METHOD M_PT100_Interpolate_Ohm2C : LREAL
VAR_INPUT
	in_lrOhm:	LREAL;	// Resistance reading [Ohm]
	// Index of the first lookup table entry with 
	// value lower than the measured resistance.
	in_nIndex:	INT;	
END_VAR
VAR
	lrR1, lrR2:	LREAL;	// Temporary variables
END_VAR
IF in_nIndex = 0 OR in_nIndex = 88	THEN
	M_PT100_Interpolate_Ohm2C	:= LookupTable[in_nIndex].celsius;
ELSE
	// Linear interpolation Example
	//	Index 8		(celsius := 	-200.0	, ohm := 	18.522	),
	//  Reading                               ohm := 	20.123
	//	Index 9		(celsius := 	-195.0	, ohm := 	20.679	),
	//
	//   TempC = -200.0 + (20.123-18.522) / (20.679-18.522) * 5.0 
	//         = -200.0 + 1.601 / 2.157 * 5.0
	//         = -196.289 degC

	lrR1	:= in_lrOhm - LookupTable[in_nIndex].ohm;
	lrR2	:= LookupTable[in_nIndex+1].ohm - LookupTable[in_nIndex].ohm;
	M_PT100_Interpolate_Ohm2C	:= LookupTable[in_nIndex].celsius + lrR1/lrR2 * lrTemStep;
END_IF
END_METHOD

// Convert raw resistance reading [bit] (Ohm*64) to degrees Celsius.
// The input value has to be devided by 64 to get the reading in [Ohm].
METHOD M_PT100_Ohm2C : LREAL
VAR_INPUT
	in_lrOhmRaw:	INT;	// Raw reading [bit]. [Ohm] = in_lrOhmRaw/64
END_VAR
VAR
	i:		INT;
	lrOhm:	LREAL; 	// PT100 Resistance reading [Ohm]
END_VAR
// Raw reading of -1 means a broken wire or failed sensor.
// The convention is to return 850 degC
IF in_lrOhmRaw	= -1	THEN
	M_PT100_Ohm2C	:= 850.0;
	RETURN;
END_IF

// Get reading in [Ohm]
lrOhm	:= INT_TO_LREAL(in_lrOhmRaw) / 64.0;


// Find the first index in the table
// where the resistance value is lower that the reading.

IF lrOhm > LookupTable[nLastIndex].ohm	THEN
	// We are increasing the index until we find a reading in the
	// table that is higher than the measurement
	FOR i := nLastIndex TO 88	DO
		IF i = 88	THEN
			// We are at the highest temperature in the lookup table.
			// Take that value;
			M_PT100_Ohm2C	:= LookupTable[i].celsius;
			RETURN;
		ELSE
			IF lrOhm < LookupTable[i].ohm	THEN
				// We crossed the correct reading.
				// Remember the index for faster next reading.
				nLastIndex	:= i-1;
				IF nLastIndex < 0	THEN
					nLastIndex	:= 0;
				END_IF
				M_PT100_Ohm2C	:= M_PT100_Interpolate_Ohm2C(lrOhm,nLastIndex);
				RETURN;
			ELSIF lrOhm = LookupTable[i].ohm	THEN
				// We crossed the correct reading.
				// Remember the index for faster next reading.
				nLastIndex	:= i;
				M_PT100_Ohm2C	:= M_PT100_Interpolate_Ohm2C(lrOhm,nLastIndex);
				RETURN;
			END_IF
		END_IF
	END_FOR
ELSIF lrOhm < LookupTable[nLastIndex].ohm	THEN
	// We are decreasing the index until we find a reading in the
	// table that is higher than the measurement
	FOR i := nLastIndex TO 0 BY  -1	DO
		IF i <= 0	THEN
			// We are at the lowest temperature in the lookup table.
			// Take that value;
			M_PT100_Ohm2C	:= LookupTable[0].celsius;
			RETURN;
		ELSE
			IF lrOhm > LookupTable[i].ohm	THEN
				// We crossed the correct reading.
				// Remember the index for faster next reading.
				nLastIndex	:= i;
				M_PT100_Ohm2C	:= M_PT100_Interpolate_Ohm2C(lrOhm,nLastIndex);
				RETURN;
			ELSIF lrOhm = LookupTable[i].ohm	THEN
				// We crossed the correct reading.
				// Remember the index for faster next reading.
				nLastIndex	:= i;
				M_PT100_Ohm2C	:= M_PT100_Interpolate_Ohm2C(lrOhm,nLastIndex);
				RETURN;
			END_IF
		END_IF
	END_FOR
ELSE
	M_PT100_Ohm2C	:= M_PT100_Interpolate_Ohm2C(lrOhm,nLastIndex);
	RETURN;
END_IF
END_METHOD

// Calculate pressure based on the status in input value
METHOD M_SetStatus
VAR_INPUT
END_VAR
VAR
END_VAR
// Set temperature sensor type
stat.nType	:= in_nType;

// Update value depending on the sensor type.
// So far, only PT100 supported.
CASE in_nType OF
	E_CRYO_SENSOR_TYPE_TEMP.PT100:
		M_SetStatus_PT100();
END_CASE
END_METHOD

// Calculate pressure based on the status in input value
METHOD M_SetStatus_PT100
VAR_INPUT
END_VAR
VAR
END_VAR
//
// Set the temperature as it is read.
// Later on we decide if it is valid or not.
//
IF NOT in_bResistor_1_64	THEN
	// Standard RTD reading
	stat.lrTempC	:= i_nValue * in_lrScale;	// Set temperature in deg C
	stat.lrTempK	:= stat.lrTempC + 273.15;	// Set temperature in deg K
ELSE	
	// RTD reading of resistance.
	// i_nValue is in [Ohm]
	stat.lrTempC	:= M_PT100_Ohm2C(i_nValue);	// Set temperature in deg C
	stat.lrTempK	:= stat.lrTempC + 273.15;	// Set temperature in deg K
END_IF

// Reading in Celsius of 850.0 means an error.
// In this case, set the Kelvin reading to 850.0 as well.
// Set error and not Valid and return.
IF stat.lrTempC = 850.0	THEN
	stat.lrTempK	:= 850.0;
	stat.bError		:= TRUE;
	stat.bValid		:= FALSE;
	RETURN;
END_IF

//
// Update validity
// Note: bInputError = (bInputUnder OR bInputOver)
//       bValid      = TRUE if PDO is OK (nothing to do with bError)
//
IF stat.bInputActive THEN
	IF stat.bInputError  AND  stat.bInputUnder  AND  in_bIgnoreUnderrange 	THEN
		// Sometimes we ignore underrange because PT100 cannot read below -200C.
		// The bUnderrange flag is still active!!!
		stat.bError	:= FALSE;
		stat.bValid	:= TRUE;
	ELSIF stat.bInputError 	THEN
		stat.bError	:= TRUE;
		stat.bValid	:= FALSE;
	ELSE
		stat.bError	:= FALSE;
		stat.bValid	:= TRUE;
	END_IF
ELSE
	stat.bError	:= TRUE;
	stat.bValid	:= FALSE;
END_IF
END_METHOD

END_FUNCTION_BLOCK

// ---- POUs/Simulation/FB_CRYO_SIM_CTRL.TcPOU
FUNCTION_BLOCK FB_CRYO_SIM_CTRL
VAR_INPUT
	in_ptr_Cryo_Ctrl:	POINTER TO FB_CRYO_CTRL;
END_VAR
VAR
	{attribute 'OPC.UA.DA' := '1'}
	SIM_Temp_Mirror:		FB_CRYO_SIM_TEMPERATURE;

	{attribute 'OPC.UA.DA' := '1'}
	SIM_Temp_LN2_Exhaust:	FB_CRYO_SIM_TEMPERATURE;
	
	{attribute 'OPC.UA.DA' := '1'}
	SIM_Temp_LN2_Inlet:		FB_CRYO_SIM_TEMPERATURE;
	
	{attribute 'OPC.UA.DA' := '1'}
	SIM_Temp_DET:			FB_CRYO_SIM_TEMPERATURE;
	
	{attribute 'OPC.UA.DA' := '1'}
	SIM_Pressure_Cryo:	FB_CRYO_SIM_PRESSURE;		// Cryo Pressure simulator
	
	{attribute 'OPC.UA.DA' := '1'}
	SIM_Pressure_Evac:	FB_CRYO_SIM_PRESSURE;		// Evacuation Pressure simulator
	
	
	
	{attribute 'OPC.UA.DA' := '1'}
	nCryoState:		E_CRYO_CTRL_STATE	:= E_CRYO_CTRL_STATE.NONE;
	{attribute 'OPC.UA.DA' := '0'}
	nCryoOldState:	E_CRYO_CTRL_STATE	:= E_CRYO_CTRL_STATE.NONE;
	
	{attribute 'OPC.UA.DA' := '0'}
	trgCMD:			R_TRIG;
	{attribute 'OPC.UA.DA' := '0'}
	trgEvacOn:		R_TRIG;
	{attribute 'OPC.UA.DA' := '0'}
	trgEvacOff:		F_TRIG;
	{attribute 'OPC.UA.DA' := '0'}
	trgInVacuum:	R_TRIG;
	{attribute 'OPC.UA.DA' := '0'}
	trgPrecoolOff:	F_TRIG;
	{attribute 'OPC.UA.DA' := '0'}
	trgCoolOff:		F_TRIG;
	{attribute 'OPC.UA.DA' := '0'}
	trgWarmupOff:	F_TRIG;
	
	nRampPeriod:	UDINT := 20000;
	
	{attribute 'OPC.UA.DA' := '0'}
	lrTmp:	LREAL;
	
	
END_VAR

//
// Get Cryo controller State
//
nCryoState	:= in_ptr_Cryo_Ctrl^.stat.nState;


//
// Execute simulators for all temperatures and pressures, etc.
//
SIM_Temp_Mirror(
	in_lrScale		:= in_ptr_Cryo_Ctrl^.Temp_Mirror.in_lrScale_1, 
	in_lrTempK		:= );
	
SIM_Temp_LN2_Exhaust(
	in_lrScale		:= in_ptr_Cryo_Ctrl^.Temp_LN2_Exhaust.in_lrScale_1, 
	in_lrTempK		:= 88.75,	//	Variation 88.75 +- 11.25, i.e. [77.50..100.00]
	in_lrTempDelta	:= 11.25,
	in_nPeriod		:= 10000,
	in_bAutoSine	:= TRUE);
	
SIM_Temp_LN2_Inlet(
	in_lrScale		:= in_ptr_Cryo_Ctrl^.Temp_LN2_Inlet.in_lrScale_1, 
	in_lrTempK		:= 77.15);
	
SIM_Temp_DET(
	in_lrScale		:= in_ptr_Cryo_Ctrl^.Temp_DET.in_lrScale_1, 
	in_lrTempK		:= );
	
SIM_Pressure_Cryo(
	in_nType		:= in_ptr_Cryo_Ctrl^.Pressure_Cryo.in_nType_1,
	in_lrBitsPerVolt:= in_ptr_Cryo_Ctrl^.Pressure_Cryo.in_lrBitsPerVolt_1, 
	in_nPeriod		:= nRampPeriod);
	
SIM_Pressure_Evac(
	in_nType		:= in_ptr_Cryo_Ctrl^.Pressure_Evac.in_nType_1,
	in_lrBitsPerVolt:= in_ptr_Cryo_Ctrl^.Pressure_Evac.in_lrBitsPerVolt_1, 
	in_nPeriod		:= nRampPeriod);


	
	
//	
// Capture Cryo controller change of state.
//
trgCMD(CLK:=(nCryoState<>nCryoOldState));
nCryoOldState	:= nCryoState;

// NOTE: This code is execute only once on each State change.
IF trgCMD.Q  THEN
	// The state of Cryo controller has changed.
	// Take action with simulators.
	CASE nCryoState OF
		
		/////////////////////////////////
		E_CRYO_CTRL_STATE.PRE_COOLING:
		/////////////////////////////////
		//
		// Trigger Bench temperature ramp 1 K below PRE_COOL threshold
		SIM_Temp_Mirror.M_RampTo(
			in_lrValueEnd	:= in_ptr_Cryo_Ctrl^.cfg.lrTemp_Precooled-1.0,
			in_nPeriod		:= nRampPeriod);

		// Trigger DET temperature ramp 1 K below PRE_COOL threshold.
		// Slow down the ramp compared to the Bench, so
		// DET temperature is slightly higher during cooldown.
		// The final temperature is the same as for the Bench.
		SIM_Temp_DET.M_RampTo(
			in_lrValueEnd	:= in_ptr_Cryo_Ctrl^.cfg.lrTemp_Precooled-1.0,
			in_nPeriod		:= nRampPeriod + 5000);
			
		/////////////////////////////////
		E_CRYO_CTRL_STATE.COOLING_DOWN:
		/////////////////////////////////
		//
		// Trigger temperature ramp 1 K below COOL threshold
		SIM_Temp_Mirror.M_RampTo(
			in_lrValueEnd	:= in_ptr_Cryo_Ctrl^.cfg.lrTemp_Cold-1.0,
			in_nPeriod		:= nRampPeriod);
			
		// Trigger temperature ramp 1 K below COOL threshold
		// Slow down the ramp compared to the Bench, so
		// DET temperature is slightly higher during cooldown.
		// The final temperature is the same as for the Bench.
		SIM_Temp_DET.M_RampTo(
			in_lrValueEnd	:= in_ptr_Cryo_Ctrl^.cfg.lrTemp_Cold-1.0,
			in_nPeriod		:= nRampPeriod + 5000);
			
		/////////////////////////////////
		E_CRYO_CTRL_STATE.WARMING_UP:
		/////////////////////////////////
		//
		// Trigger temperature ramp to in_ptr_Cryo_Ctrl^.cfg.lrTemp_Warm (~10C)
		SIM_Temp_Mirror.M_RampTo(
			in_lrValueEnd	:= in_ptr_Cryo_Ctrl^.cfg.lrTemp_Warm + 1.0,
			in_nPeriod		:= nRampPeriod);
			
			
		// Trigger temperature ramp to in_ptr_Cryo_Ctrl^.cfg.lrTemp_Warm (~10C)
		// Speed up the ramp compared to the Bench, so
		// DET temperature is slightly higher during warm-up.
		// The final temperature is the same as for the Bench.
		SIM_Temp_DET.M_RampTo(
			in_lrValueEnd	:= in_ptr_Cryo_Ctrl^.cfg.lrTemp_Warm + 1.0,
			in_nPeriod		:= nRampPeriod - 2000);
			
		/////////////////////////////////
		E_CRYO_CTRL_STATE.REPRESSURIZING:
		/////////////////////////////////
		//
		// Trigger Cryo vacuum ramp to atmospheric pressure ~820 mbar
		SIM_Pressure_Cryo.M_RampTo(
			in_lrValueEnd	:= 820.0,
			in_nPeriod		:= 17000);
			
		// Follow the same ramp with Evac but a bit slower.
		SIM_Pressure_Evac.M_RampTo(
			in_lrValueEnd	:= 820.0,
			in_nPeriod		:= 20000);
	END_CASE

END_IF


//
// Evacuation Pressure simulation
//
// Capture Evacuation ON/OFF trigger
trgEvacOn(CLK := in_ptr_Cryo_Ctrl^.ctrl.bEnable_Evac);
trgEvacOff(CLK := in_ptr_Cryo_Ctrl^.ctrl.bEnable_Evac);
IF	trgEvacOn.Q THEN
	// Trigger vacuum ramp 0.0001 mbar below Good Vacuum
	SIM_Pressure_Cryo.M_StartCurve(
		in_lrValueEnd	:= in_ptr_Cryo_Ctrl^.Pressure_Cryo.in_lrLimitGoodVac - 0.0001, 
		in_nPeriod		:= 20000, 
		in_lrCurveScale	:= 0.3);
ELSIF trgEvacOff.Q THEN
	// Evacuation stopped.
	// Keep the pressure as it is.
	SIM_Pressure_Cryo.M_Stop();
END_IF


//
// If Turbo Pump is running, keep Evacuation pressure 1.0e-05 below the Cryo pressure.
// Value is calculated on every cycle.
//
IF in_ptr_Cryo_Ctrl^.EvacSys.stat.bTurboPumpON THEN
	SIM_Pressure_Evac.M_SetValue(SIM_Pressure_Cryo.lrPress - 1.0E-05);
END_IF


//
// To get more realistic evacuation,
// Restart simulated curve when inVacuum is triggered.
//
//trgInVacuum(CLK := in_ptr_Cryo_Ctrl^.Pressure_Cryo.stat.bInVacuum);
trgInVacuum(CLK := in_ptr_Cryo_Ctrl^.stat.bInVacuum);
IF trgInVacuum.Q THEN
	SIM_Pressure_Cryo.M_StartCurve(
		in_lrValueEnd	:= in_ptr_Cryo_Ctrl^.Pressure_Cryo.in_lrLimitGoodVac - 0.0001, 
		in_nPeriod		:= 10000, 
		in_lrCurveScale	:= 0.3);
END_IF

			
//
// Capture events when buttons are released 
// and temperature transitions interrupted.
//

// Capture pre-cooling, cooling or warmup button release.
// Stop ramping in that case.
trgPrecoolOff	(CLK:=in_ptr_Cryo_Ctrl^.ctrl.bEnable_Precool);
trgCoolOff		(CLK:=in_ptr_Cryo_Ctrl^.ctrl.bEnable_Cool);
trgWarmupOff	(CLK:=in_ptr_Cryo_Ctrl^.ctrl.bEnable_Warmup);

IF	trgPrecoolOff.Q OR trgCoolOff.Q OR trgWarmupOff.Q	THEN
	SIM_Temp_Mirror.M_Stop();
	SIM_Temp_DET.M_Stop();
END_IF

END_FUNCTION_BLOCK

// ---- POUs/Simulation/FB_CRYO_SIM_TEMPERATURE.TcPOU
//
// This FB simulates temperature in degK.
//
FUNCTION_BLOCK FB_CRYO_SIM_TEMPERATURE
VAR_INPUT
	in_lrScale:		LREAL 	:= 0.1;		// Scale factor, T = raw * scale. Default 0.1
	in_lrTempK:		LREAL	:= 283.15;	// Start Temperature [K]
	in_lrTempDelta:	LREAL	:= 11.25;	// Delta Temperature +- for SINE wave [K]
	in_nPeriod:		UDINT	:= 10000;	// RAMP/SINE Command period, default 10000ms = 10s
	in_bAutoSine:	BOOL	:= FALSE;	// Flag if SINE wave should start immediately
	
END_VAR
VAR
	q_nStatus	AT%Q*:	UINT	:= 0;	// Simulated status
	q_nValue	AT%Q*:	INT		:= 100;	// Simulated value [bit]
	
	{attribute 'OPC.UA.DA' := '0'}
	bStarted:		BOOL := FALSE;
	{attribute 'OPC.UA.DA' := '0'}
	toggleTimer:	TON;		// Timer for PDO (alive) toggle
	{attribute 'OPC.UA.DA' := '0'}
	rampTimer:		TON;		// Timer for temperature ramp

	{attribute 'OPC.UA.DA' := '0'}
	nToggleMask:	UINT := 2#1000_0000_0000_0000;

	lrTempK:		LREAL	:= 283.15;	// Simulated temperature [K]
	{attribute 'OPC.UA.DA' := '0'}
	lrTempStart:	LREAL	:= 283.15;	// Simulated temperature start [K]
	{attribute 'OPC.UA.DA' := '0'}
	lrTempEnd:		LREAL	:= 0.0;		// Simulated temperature end   [K]
	{attribute 'OPC.UA.DA' := '0'}
	lrTempDelta:	LREAL	:= 11.25;	// Delta Temperature +- for SINE wave [K]
	{attribute 'OPC.UA.DA' := '0'}
	nValue:			INT		:= 100;		// Simulated value [bit]

	{attribute 'OPC.UA.DA' := '0'}
	nPeriod:		UDINT	:= 10000;	// RAMP/SINE Command period, default 10000ms = 10s
	
	{attribute 'OPC.UA.DA' := '0'}
	nState:		INT	:= SIM_TEMP_STATE_FIXED;
	
END_VAR
VAR CONSTANT 
	{attribute 'OPC.UA.DA' := '0'}
    SIM_TEMP_STATE_NONE:	INT :=  0;
	{attribute 'OPC.UA.DA' := '0'}
    SIM_TEMP_STATE_FIXED:	INT := 10;
	{attribute 'OPC.UA.DA' := '0'}
    SIM_TEMP_STATE_RAMP:	INT := 20;
	{attribute 'OPC.UA.DA' := '0'}
    SIM_TEMP_STATE_SINE:	INT := 30;
	
	{attribute 'OPC.UA.DA' := '0'}
    SIM_TEMP_RAMP_UP:		INT := 0;
	{attribute 'OPC.UA.DA' := '0'}
    SIM_TEMP_RAMP_DOWN:		INT := 1;
	
END_VAR

//
// Simulate terminal alive toggle every 160ms.
//
IF NOT bStarted THEN
	bStarted	:= TRUE;
	lrTempK		:= in_lrTempK;	// Assign starting value
	lrTempDelta	:= in_lrTempDelta;
	nPeriod		:= in_nPeriod;
	IF in_bAutoSine THEN
		M_StartSine(in_lrValueStart:=lrTempK,
					in_lrValueDelta:=lrTempDelta,
					in_nPeriod:=nPeriod);
	END_IF
	toggleTimer(IN:=FALSE);
END_IF
toggleTimer(IN:=TRUE,PT:=T#160MS);

IF toggleTimer.Q THEN
	q_nStatus	:= q_nStatus XOR nToggleMask;
	// Restart the timer
	toggleTimer(IN:=FALSE);
END_IF


//
// Handle states 
//
IF nState = SIM_TEMP_STATE_RAMP THEN
	rampTimer(IN:=TRUE);
	lrTempK	:=	lrTempStart + 
				(lrTempEnd - lrTempStart)* TIME_TO_LREAL(rampTimer.ET)/TIME_TO_LREAL(rampTimer.PT);
	IF rampTimer.Q THEN
		rampTimer(IN:=FALSE);
		nState	:= SIM_TEMP_STATE_FIXED;
	END_IF
ELSIF nState = SIM_TEMP_STATE_SINE THEN
	rampTimer(IN:=TRUE);
	lrTempK	:=	lrTempStart + 
				lrTempDelta * SIN(2 * PI * TIME_TO_LREAL(rampTimer.ET)/TIME_TO_LREAL(rampTimer.PT));
	IF rampTimer.Q THEN
		rampTimer(IN:=FALSE);
		// Continue with the sine wave.
		rampTimer(IN:=TRUE,PT:=UDINT_TO_TIME(nPeriod));
	END_IF
END_IF



//
// Set the raw reading, i.e. K -> bit.
//
q_nValue	:= M_degK2bit(lrTempK);

METHOD M_bit2degK : LREAL
VAR_INPUT
	in_nValue:	INT;
END_VAR
//
// Set the raw reading, i.e. K -> bit.
// Conversion is K -> C -> bit.
//
M_bit2degK	:= in_nValue * in_lrScale + 273.15;
END_METHOD

METHOD M_degK2bit : INT
VAR_INPUT
	in_lrValue:	LREAL;
END_VAR
//
// Set the raw reading, i.e. K -> bit.
// Conversion is K -> C -> bit.
//
M_degK2bit	:= LREAL_TO_INT((in_lrValue - 273.15) / in_lrScale);
END_METHOD

METHOD M_RampTo
VAR_INPUT
	in_lrValueEnd:		LREAL;
	in_nPeriod:			UDINT	:= 10000;	// RAMP/SINE Command period, default 10000ms = 10s
END_VAR
rampTimer(IN:=FALSE);
rampTimer(IN:=TRUE,PT:=UDINT_TO_TIME(in_nPeriod));
lrTempStart	:= lrTempK;
lrTempEnd	:= in_lrValueEnd;
nPeriod		:= in_nPeriod;
nState		:= SIM_TEMP_STATE_RAMP;
END_METHOD

METHOD M_SetValue
VAR_INPUT
	in_lrValue:	LREAL;
END_VAR
rampTimer(IN:=FALSE);
lrTempK	:= in_lrValue;
nState	:= SIM_TEMP_STATE_FIXED;
END_METHOD

METHOD M_StartRamp
VAR_INPUT
	in_lrValueStart:	LREAL;
	in_lrValueEnd:		LREAL;
	in_nPeriod:			UDINT	:= 10000;	// RAMP/SINE Command period, default 10000ms = 10s
END_VAR
rampTimer(IN:=FALSE);
rampTimer(IN:=TRUE,PT:=UDINT_TO_TIME(in_nPeriod));
lrTempStart	:= in_lrValueStart;
lrTempEnd	:= in_lrValueEnd;
nPeriod		:= in_nPeriod;
nState		:= SIM_TEMP_STATE_RAMP;
END_METHOD

METHOD M_StartSine
VAR_INPUT
	in_lrValueStart:	LREAL;
	in_lrValueDelta:	LREAL;
	in_nPeriod:			UDINT	:= 10000;	// RAMP/SINE Command period, default 10000ms = 10s
END_VAR
rampTimer(IN:=FALSE);
rampTimer(IN:=TRUE,PT:=UDINT_TO_TIME(in_nPeriod));
lrTempStart	:= in_lrValueStart;
lrTempDelta	:= in_lrValueDelta;
nPeriod		:= in_nPeriod;
nState		:= SIM_TEMP_STATE_SINE;
END_METHOD

METHOD M_Stop
VAR_INPUT
END_VAR
// Stop ramping.
// Keep value as it is.
rampTimer(IN:=FALSE);
nState	:= SIM_TEMP_STATE_FIXED;
END_METHOD

END_FUNCTION_BLOCK

// ---- POUs/Simulation/FB_CRYO_SIM_PRESSURE.TcPOU
//
// This FB simulates pressure.
//
FUNCTION_BLOCK FB_CRYO_SIM_PRESSURE
VAR_INPUT
	in_nType:	E_CRYO_SENSOR_TYPE_PRESS;
	// Scale factor bits -> Volt, U = raw / scale. 
	// Default for 16-bit, +-10V or 0..10V AI: 2^16/10/2 = 3276.8 bit
	in_lrBitsPerVolt:	LREAL := 3276.8;	// Scale factor, U = raw / scale. Default 3276.8
	in_lrPress:		LREAL	:= 777.0;	// Starting Pressure
	in_nPeriod:		UDINT	:= 10000;	// RAMP Command period, default 10000ms = 10s
	
END_VAR
VAR
	q_nStatus	AT%Q*:	UINT	:= 0;		// Simulated status
	q_nValue	AT%Q*:	INT		:= 27953;	// Simulated value [bit] = 777 mbar
	
	{attribute 'OPC.UA.DA' := '0'}
	bStarted:		BOOL := FALSE;
	{attribute 'OPC.UA.DA' := '0'}
	toggleTimer:	TON;		// Timer for PDO (alive) toggle
	{attribute 'OPC.UA.DA' := '0'}
	rampTimer:		TON;		// Timer for temperature ramp

	{attribute 'OPC.UA.DA' := '0'}
	nToggleMask:	UINT := 2#1000_0000_0000_0000;

	lrPress:		LREAL	:= 777.0;	// Simulated Pressure
	{attribute 'OPC.UA.DA' := '0'}
	lrPressStart:	LREAL	:= 0.0;		// Simulated Pressure start[mbar]
	{attribute 'OPC.UA.DA' := '0'}
	lrPressEnd:		LREAL	:= 0.0;		// Simulated Pressure end  [mbar]
	{attribute 'OPC.UA.DA' := '0'}
	lrPressDelta:	LREAL	:= 0.0;		// Simulated Pressure delta for curve  [mbar]
	{attribute 'OPC.UA.DA' := '0'}
	lrCurveScale:	LREAL	:= 0.3;		// t^lrCurveScale factor
	{attribute 'OPC.UA.DA' := '0'}
	nValue:			INT		:= 27953;	// Simulated value [bit]
	{attribute 'OPC.UA.DA' := '0'}
	nPeriod:		UDINT	:= 10000;	// RAMP Command period, default 10000ms = 10s
	
	{attribute 'OPC.UA.DA' := '0'}
	State:		INT	:= SIM_VACUUM_STATE_FIXED;
	
	// Temporary variables
	{attribute 'OPC.UA.DA' := '0'}
	lrTmp1:		LREAL;
	
END_VAR
VAR CONSTANT 
	{attribute 'OPC.UA.DA' := '0'}
    SIM_VACUUM_STATE_NONE:	INT :=  0;
	{attribute 'OPC.UA.DA' := '0'}
    SIM_VACUUM_STATE_FIXED:	INT := 10;
	{attribute 'OPC.UA.DA' := '0'}
    SIM_VACUUM_STATE_RAMP:	INT := 20;
	{attribute 'OPC.UA.DA' := '0'}
    SIM_VACUUM_STATE_CURVE:	INT := 30;
	
	{attribute 'OPC.UA.DA' := '0'}
    SIM_VACUUM_RAMP_UP:		INT := 0;
	{attribute 'OPC.UA.DA' := '0'}
    SIM_VACUUM_RAMP_DOWN:	INT := 1;
	
END_VAR

//
// Simulate terminal alive toggle every 160ms.
//
IF NOT bStarted THEN
	bStarted	:= TRUE;
	lrPress		:= in_lrPress;
	nPeriod		:= in_nPeriod;
	toggleTimer(IN:=FALSE);
END_IF
toggleTimer(IN:=TRUE,PT:=T#160MS);

IF toggleTimer.Q THEN
	q_nStatus	:= q_nStatus XOR nToggleMask;
	// Restart the timer
	toggleTimer(IN:=FALSE);
END_IF



//
// Handle states
//
rampTimer(IN:=TRUE);
IF State = SIM_VACUUM_STATE_RAMP THEN
	lrPress	:=	lrPressStart + 
				(lrPressEnd - lrPressStart)* TIME_TO_LREAL(rampTimer.ET)/TIME_TO_LREAL(rampTimer.PT);
	IF rampTimer.Q THEN
		rampTimer(IN:=FALSE);
		State	:= SIM_VACUUM_STATE_FIXED;
	END_IF
ELSIF State = SIM_VACUUM_STATE_CURVE THEN
	lrTmp1	:= TIME_TO_LREAL(rampTimer.ET)/TIME_TO_LREAL(rampTimer.PT);
	lrTmp1	:= EXPT(lrTmp1,lrCurveScale);
	lrPress	:=	lrPressStart + (lrPressEnd - lrPressStart)* lrTmp1;
	IF rampTimer.Q THEN
		rampTimer(IN:=FALSE);
		State	:= SIM_VACUUM_STATE_FIXED;
	END_IF
END_IF


//
// Set the raw reading, i.e. mbar -> bit.
// Conversion is mbar -> Volt -> bit.
//
IF lrPress > 0.0  THEN
	q_nValue	:= M_mbar2bit(lrPress);
END_IF

METHOD M_bit2mbar : LREAL
VAR_INPUT
	in_nBits:	INT;
END_VAR
VAR
	lrVoltage:	LREAL;
	lrPressure:	LREAL;
END_VAR
lrVoltage	:= in_nBits / in_lrBitsPerVolt;

CASE in_nType OF 
	E_CRYO_SENSOR_TYPE_PRESS.PKR_250,
	E_CRYO_SENSOR_TYPE_PRESS.PKR_360:
		// Conversion Volt -> mbar.
		// Pfeiffer PKR250/251
		// P = 10^(C1 * U - C2).
		// C1 = 1.667, C2 = d = 11.33
		// P = 10^(1.667 * U - 11.33)
		// U = (log(P)+C2)/C1
		// U = (log(P)+11.33)/1.667
		lrPressure	:= EXPT(10.0, (1.667 * lrVoltage - 11.33));
	E_CRYO_SENSOR_TYPE_PRESS.CMR_361:
		// Conversion Volt -> mbar.
		// Pfeiffer CMR361
		// P = (U - 1) * C1 * C2 [mbar]
		// C1 = 0.125, C2=FullScale = 1000 
		// P = (U - 1) * 0.125 * 1000.0 = (U-1) * 125[mbar]
		// P = (U-1) * 125
		// U = P/125 + 1
		lrPressure	:= (lrVoltage - 1) * 125;
	E_CRYO_SENSOR_TYPE_PRESS.WRG_D_NW25:
		// Edwards WRG-D-NW25 Conversion Volt -> mbar.
		// Range 10^-9 .. 100
		// P = 10^(C1 * U - C2).
		// P = 10^(1.5 * U - 12.0)
		// Valid range for U is 2.0-10.0
		lrPressure	:= EXPT(10.0, (1.5 * lrVoltage - 12.0));
END_CASE

M_bit2mbar	:= lrPressure;
END_METHOD

METHOD M_mbar2bit : INT
VAR_INPUT
	in_lrValue:	LREAL;
END_VAR
VAR
	lrValue:	LREAL;
	lrVoltage:	LREAL;
END_VAR
// Pressure cannot be zero
lrValue := MAX(1.0E-9,in_lrValue);

CASE in_nType OF 
	E_CRYO_SENSOR_TYPE_PRESS.PKR_250,
	E_CRYO_SENSOR_TYPE_PRESS.PKR_360:
		// Conversion Volt -> mbar.
		// Pfeiffer PKR250/251
		// P = 10^(C1 * U - C2).
		// C1 = 1.667, C2 = d = 11.33
		// P = 10^(1.667 * U - 11.33)
		// U = (log(P)+C2)/C1
		// U = (log(P)+11.33)/1.667
		lrVoltage	:= (LOG(lrValue) + 11.33) / 1.667;
	E_CRYO_SENSOR_TYPE_PRESS.CMR_361:
		// Conversion Volt -> mbar.
		// Pfeiffer CMR361
		// P = (U - 1) * C1 * C2 [mbar]
		// C1 = 0.125, C2=FullScale = 1000 
		// P = (U - 1) * 0.125 * 1000.0 = (U-1) * 125[mbar]
		// P = (U-1) * 125
		// U = P/125 + 1
		lrVoltage	:= lrValue/125 + 1.0;
	E_CRYO_SENSOR_TYPE_PRESS.WRG_D_NW25:
		// Edwards WRG-D-NW25 Conversion Volt -> mbar.
		// Range 10^-9 .. 100
		// P = 10^(C1 * U - C2).
		// P = 10^(1.5 * U - 12.0)
		// Valid range for U is 2.0-10.0
		lrVoltage	:= (LOG(lrValue) + 12.0) / 1.5;
END_CASE

M_mbar2bit	:= LREAL_TO_INT(lrVoltage * in_lrBitsPerVolt);
END_METHOD

METHOD M_RampTo
VAR_INPUT
	in_lrValueEnd:		LREAL;
	in_nPeriod:			UDINT	:= 10000;	// RAMP/SINE Command period, default 10000ms = 10s
END_VAR
rampTimer(IN:=FALSE);
rampTimer(IN:=TRUE,PT:=UDINT_TO_TIME(in_nPeriod));
lrPressStart	:= lrPress;
lrPressEnd		:= in_lrValueEnd;
nPeriod			:= in_nPeriod;
State			:= SIM_VACUUM_STATE_RAMP;
END_METHOD

METHOD M_SetValue
VAR_INPUT
	in_lrValue:	LREAL;
END_VAR
rampTimer(IN:=FALSE);
lrPress	:= in_lrValue;
State	:= SIM_VACUUM_STATE_FIXED;
END_METHOD

METHOD M_StartCurve
VAR_INPUT
	in_lrValueEnd:		LREAL;
	in_nPeriod:			UDINT	:= 20000;	// RAMP/SINE Command period, default 10000ms = 10s
	in_lrCurveScale:	LREAL	:= 0.3;		// t^lrCurveScale factor
END_VAR
rampTimer(IN:=FALSE);
rampTimer(IN:=TRUE,PT:=UDINT_TO_TIME(in_nPeriod));
lrPressStart	:= lrPress;
lrPressEnd		:= in_lrValueEnd;
lrCurveScale	:= in_lrCurveScale;
State			:= SIM_VACUUM_STATE_CURVE;
END_METHOD

METHOD M_StartRamp
VAR_INPUT
	in_lrValueStart:	LREAL;
	in_lrValueEnd:		LREAL;
END_VAR
rampTimer(IN:=FALSE);
rampTimer(IN:=TRUE,PT:=UDINT_TO_TIME(nPeriod));
lrPressStart	:= in_lrValueStart;
lrPressEnd		:= in_lrValueEnd;
State			:= SIM_VACUUM_STATE_RAMP;
END_METHOD

METHOD M_Stop
VAR_INPUT
END_VAR
// Stop ramping.
// Keep value as it is.
rampTimer(IN:=FALSE);
State	:= SIM_VACUUM_STATE_FIXED;
END_METHOD

END_FUNCTION_BLOCK

// ---- POUs/Sensors/FB_CRYO_PRESSURE_VOTE.TcPOU
//
// This FB calculates resulting pressure applying the selected voting method.
// Up to five pressure sensors are used in the calculation.
// The resulting value is a combination of values from available/valid sensors.
// For more info, see method M_SetStatus().
//
FUNCTION_BLOCK FB_CRYO_PRESSURE_VOTE
VAR_INPUT
	{attribute 'OPC.UA.DA' := '0'}
	in_bSimulation:	BOOL	:= FALSE;	// If TRUE, the pressure value is simulated.
	
	{attribute 'OPC.UA.DA' := '0'}
	in_nNumSensor:	INT;				// Number of sensors used by voiting method.
	
	{attribute 'OPC.UA.DA' := '0'}
	in_nVoteMethod:	E_CRYO_VOTE	:= E_CRYO_VOTE.V_AVE;	// Active voting method.
	
	// Five pointers to instances of FB_CRYO_SENSOR_PRESSURE.
	// Pointers should only be set to existing pressure sensors.
	{attribute 'OPC.UA.DA' := '0'}
	in_pSensor1:		POINTER TO FB_CRYO_SENSOR_PRESSURE	:= 0;
	{attribute 'OPC.UA.DA' := '0'}
	in_pSensor2:		POINTER TO FB_CRYO_SENSOR_PRESSURE	:= 0;
	{attribute 'OPC.UA.DA' := '0'}
	in_pSensor3:		POINTER TO FB_CRYO_SENSOR_PRESSURE	:= 0;
	{attribute 'OPC.UA.DA' := '0'}
	in_pSensor4:		POINTER TO FB_CRYO_SENSOR_PRESSURE	:= 0;
	{attribute 'OPC.UA.DA' := '0'}
	in_pSensor5:		POINTER TO FB_CRYO_SENSOR_PRESSURE	:= 0;

END_VAR
VAR
	{attribute 'OPC.UA.DA' := '1'}
	stat:		T_CRYO_PRESSURE_VOTE_STATUS;	// Complete status
	
	pSensor:	ARRAY [1..5] OF POINTER TO FB_CRYO_SENSOR_PRESSURE;
END_VAR

// If not configured yet, return.
IF NOT M_Configure()	THEN
	RETURN;
END_IF

// Set warnings for sensors with problems
M_CheckWarnings();

// Set the calculated vacuum pressure
M_SetStatus();

METHOD M_CheckWarnings : BOOL
VAR_INPUT
END_VAR
VAR
	i:			INT;
END_VAR
FOR i:=1 TO in_nNumSensor DO
	IF pSensor[i] <> 0  THEN
		// The set pointer (<> 0) indicates that the sensor is connected.
		// Warnings could be set only for connected sensors.
		IF  pSensor[i]^.stat.bValid	THEN
			// Clear warning
			M_SetWarning(i, FALSE);
		ELSE
			// Set warning
			M_SetWarning(i, TRUE);
		END_IF
	ELSE
		// Not connected sensors don't have warnings
		M_SetWarning(i, FALSE);
	END_IF
END_FOR
END_METHOD

METHOD M_Configure : BOOL
VAR_INPUT
END_VAR
VAR
	j:					INT;
END_VAR
VAR_INST
	{attribute 'OPC.UA.DA' := '0'}
	i:	INT := 0;
	{attribute 'OPC.UA.DA' := '0'}
	bConfigured:	BOOL := FALSE;
END_VAR
// The number of sensors must be between 1 and 5.
IF in_nNumSensor < 1 OR in_nNumSensor > 5 THEN
	// Set error string
	stat.sStatus	:= 'ERROR: Number of sensors (var in_nNumSensor) is not in range [1..5]';
	RETURN;
END_IF

// Configure the system in stages after boot-up.
// WARNING:
// It seems that setting of pointers takes some time and cannot be done in FB_Init.
// After 40 cycles, we set pointers to sensors.
// After 80 cycles, we set general configuration parameters and complete configuration.
IF NOT bConfigured THEN
	i	:= i + 1;
	IF i = 40 THEN
		// Assign pointers to the sensor device instances
		pSensor[1] := in_pSensor1;
		pSensor[2] := in_pSensor2;
		pSensor[3] := in_pSensor3;
		pSensor[4] := in_pSensor4;
		pSensor[5] := in_pSensor5;
	ELSIF i >= 80 THEN
		FOR j := 1 TO in_nNumSensor DO
			IF pSensor[j] <> 0 THEN
				// Set the status flag that the sensor is connected.
				M_SetConnected(j, TRUE);
				// At least one pointer is not zero.
				// We have finished configuration.
				bConfigured	:= TRUE;
			ELSE
				M_SetConnected(j, FALSE);
			END_IF
		END_FOR
	END_IF
END_IF

M_Configure	:= bConfigured;
END_METHOD

METHOD M_SetConnected : BOOL
VAR_INPUT
	in_nIndex:		INT;
	in_bConnected:	BOOL;
END_VAR
CASE in_nIndex OF
	1:
		stat.bConnSens1	:= in_bConnected;
	2:
		stat.bConnSens2	:= in_bConnected;
	3:
		stat.bConnSens3	:= in_bConnected;
	4:
		stat.bConnSens4	:= in_bConnected;
	5:
		stat.bConnSens5	:= in_bConnected;
END_CASE
END_METHOD

// Calculate pressure based on the status of the two sensors
METHOD M_SetStatus
VAR_INPUT
END_VAR
VAR
	lrTmp:		LREAL;	// Temporary var
	nSample:	INT;
	i:			INT;
END_VAR
//
// If simulated, set the simulated value and return.
//
IF in_bSimulation THEN
	stat.bSimulated	:= TRUE;
	stat.bValid		:= TRUE;
	stat.lrPressure	:= stat.lrSimPressure;
	RETURN;
ELSE
	stat.bSimulated	:= FALSE;
END_IF


//
// Get the pressure depending on the voting method.
//
CASE in_nVoteMethod OF
	E_CRYO_VOTE.V_AVE:
		M_SetStatus_Average();
	E_CRYO_VOTE.V_MIN:
		M_SetStatus_Minimum();
	E_CRYO_VOTE.V_MAX:
		M_SetStatus_Maximum();
	E_CRYO_VOTE.V_1oo2:
		M_SetStatus_FirstValid();
	E_CRYO_VOTE.V_2oo3:
		M_SetStatus_XooY(2,3);
	E_CRYO_VOTE.V_3oo5:
		M_SetStatus_XooY(3,5);
ELSE
	;
END_CASE


//
// If the reading is valid, set the simulated value to it.
// This way, switching from normal to simulation will result in
// no jump in the value.
//
IF stat.bValid  THEN
	stat.lrSimPressure	:= stat.lrPressure;
END_IF
END_METHOD

// Calculate pressure based on the average of all valid sensor readings
METHOD M_SetStatus_Average
VAR_INPUT
END_VAR
VAR
	lrTmp:		LREAL;	// Temporary var for sum of pressures
	nSample:	INT;	// Number of valid sensor readings
	i:			INT;
END_VAR
lrTmp	:= 0.0;
nSample	:= 0;
FOR i:=1 TO in_nNumSensor DO
	IF pSensor[i] <> 0  THEN
		IF  pSensor[i]^.stat.bValid	THEN
			lrTmp	:= lrTmp + pSensor[i]^.stat.lrPressure;
			nSample	:= nSample + 1;
		END_IF
	END_IF
END_FOR
IF nSample > 0	THEN
	stat.lrPressure	:= lrTmp / nSample;
	stat.bValid		:= TRUE;
ELSE
	stat.lrPressure	:= 9999;
	stat.bValid		:= FALSE;
END_IF
END_METHOD

// Calculate pressure based on the first measured valid value
METHOD M_SetStatus_FirstValid
VAR_INPUT
END_VAR
VAR
	lrTmp:		LREAL;	// Temporary var for sum of pressures
	nSample:	INT;	// Number of valid sensor readings
	i:			INT;
END_VAR
nSample	:= 0;
FOR i:=1 TO in_nNumSensor DO
	IF pSensor[i] <> 0  THEN
		IF  pSensor[i]^.stat.bValid	THEN
			lrTmp	:= pSensor[i]^.stat.lrPressure;
			nSample	:= nSample + 1;
			EXIT;
		END_IF
	END_IF
END_FOR
IF nSample > 0	THEN
	stat.lrPressure	:= lrTmp;
	stat.bValid		:= TRUE;
ELSE
	stat.lrPressure	:= 9999;
	stat.bValid		:= FALSE;
END_IF
END_METHOD

// Calculate pressure based on the highest measured valid value
METHOD M_SetStatus_Maximum
VAR_INPUT
END_VAR
VAR
	lrTmp:		LREAL;	// Temporary var for sum of pressures
	nSample:	INT;	// Number of valid sensor readings
	i:			INT;
END_VAR
lrTmp	:= -100000.0;	// Dummy starting value
nSample	:= 0;
FOR i:=1 TO in_nNumSensor DO
	IF pSensor[i] <> 0  THEN
		IF  pSensor[i]^.stat.bValid	THEN
			IF pSensor[i]^.stat.lrPressure > lrTmp THEN
				lrTmp	:= pSensor[i]^.stat.lrPressure;
			END_IF
			nSample	:= nSample + 1;
		END_IF
	END_IF
END_FOR
IF nSample > 0	THEN
	stat.lrPressure	:= lrTmp;
	stat.bValid		:= TRUE;
ELSE
	stat.lrPressure	:= 9999;
	stat.bValid		:= FALSE;
END_IF
END_METHOD

// Calculate pressure based on the lowest measured valid value
METHOD M_SetStatus_Minimum
VAR_INPUT
END_VAR
VAR
	lrTmp:		LREAL;	// Temporary var for sum of pressures
	nSample:	INT;	// Number of valid sensor readings
	i:			INT;
END_VAR
lrTmp	:= 100000.0;	// Dummy starting value
nSample	:= 0;
FOR i:=1 TO in_nNumSensor DO
	IF pSensor[i] <> 0  THEN
		IF  pSensor[i]^.stat.bValid	THEN
			IF pSensor[i]^.stat.lrPressure < lrTmp THEN
				lrTmp	:= pSensor[i]^.stat.lrPressure;
			END_IF
			nSample	:= nSample + 1;
		END_IF
	END_IF
END_FOR
IF nSample > 0	THEN
	stat.lrPressure	:= lrTmp;
	stat.bValid		:= TRUE;
ELSE
	stat.lrPressure	:= 9999;
	stat.bValid		:= FALSE;
END_IF
END_METHOD

// Calculate pressure based on the status of the two sensors
METHOD M_SetStatus_XooY
VAR_INPUT
	in_nNum:	INT;	// Number of readings to select for voting (X)
	in_nTotal:	INT;	// Total number of readings to check (Y)
END_VAR
VAR
	idx_i, idx_j:	INT;
	nTmp:		INT;			// Temporary INT var
	lrTmp:		LREAL	:= 0.0;	// Temporary var for sum of pressures
	nValid:		INT		:= 0;	// Total number of valid readings
	nSample:	INT		:= 0;	// Number of valid sensor readings
	
	aDiff:		ARRAY [1..5,1..5] OF LREAL;	// Table of absolute differences
	aDiffSum:	ARRAY [1..5] OF LREAL;		// Array of sums of absolute differences
	// Array of indexes of sums of absolute differences
	aDiffSumIdx:ARRAY [1..5] OF INT := [1,2,3,4,5];		
	lrAbsDiff:	LREAL;						// Absolute difference between two readings
	
	i:			INT;
	j:			INT;
END_VAR
//
//	Get the number of valid readings and calculate the average
//
FOR i:=1 TO in_nTotal DO
	IF pSensor[i] <> 0  THEN
		IF  pSensor[i]^.stat.bValid	THEN
			lrTmp	:= lrTmp + pSensor[i]^.stat.lrPressure;
			nValid	:= nValid + 1;
		END_IF
	END_IF
END_FOR


//
// Vote X out of Y
//
IF nValid >= in_nNum	THEN
	//
	// Calculate relative differences between two readings, 
	// relative to the bigger ABS value.
	// Table is symetric. Calculate only the half (triangle) on the right. 
	// Make a copy to the other half.
	//
	FOR i:=1 TO in_nTotal DO
		FOR j:=i+1 TO in_nTotal DO
			IF pSensor[i] <> 0  AND  pSensor[j] <> 0	THEN
				IF pSensor[i]^.stat.bValid  AND  pSensor[j]^.stat.bValid	THEN
					lrAbsDiff	:= ABS(pSensor[i]^.stat.lrPressure - pSensor[j]^.stat.lrPressure);
					aDiff[i,j]	:= lrAbsDiff;
					aDiff[j,i]	:= lrAbsDiff;
				ELSE
					aDiff[i,j]	:= 9999.0;
					aDiff[j,i]	:= 9999.0;
				END_IF
			ELSE
				aDiff[i,j]	:= 9999.0;
				aDiff[j,i]	:= 9999.0;
			END_IF
		END_FOR
	END_FOR

	//
	// Get the sum of all differences for each reading.
	//
	FOR i:=1 TO in_nTotal DO
		aDiffSum[i]	:= 0.0;
		FOR j:=1 TO in_nTotal DO
			aDiffSum[i]	:= aDiffSum[i] + aDiff[i,j];
		END_FOR
	END_FOR

	//
	// Sort the indexes for differences in accending order (low sum first).
	//
	FOR i:=1 TO in_nTotal DO
		FOR j:=i+1 TO in_nTotal DO
			idx_i	:= aDiffSumIdx[i];
			idx_j	:= aDiffSumIdx[j];
			IF aDiffSum[idx_j] < aDiffSum[idx_i]	THEN
				// Swap indexes
				nTmp			:= aDiffSumIdx[j];
				aDiffSumIdx[j]	:= aDiffSumIdx[i];
				aDiffSumIdx[i]	:= nTmp;
			END_IF
		END_FOR
	END_FOR

	
	//					
	// Get the average of selected in_nNum readings.
	// Assign the result to the pressure.
	//
	lrTmp	:= 0.0;
	FOR i:=1 TO in_nNum DO
		idx_i	:= aDiffSumIdx[i];
		lrTmp	:= lrTmp + pSensor[idx_i]^.stat.lrPressure;
	END_FOR
	
	stat.lrPressure	:= lrTmp / in_nNum;
	stat.bValid		:= TRUE;
ELSE
	stat.lrPressure	:= 9999;
	stat.bValid		:= FALSE;
END_IF
END_METHOD

METHOD M_SetWarning : BOOL
VAR_INPUT
	in_nIndex:		INT;
	in_bWarning:	BOOL;
END_VAR
CASE in_nIndex OF
	1:
		stat.bWarnSens1	:= in_bWarning;
	2:
		stat.bWarnSens2	:= in_bWarning;
	3:
		stat.bWarnSens3	:= in_bWarning;
	4:
		stat.bWarnSens4	:= in_bWarning;
	5:
		stat.bWarnSens5	:= in_bWarning;
END_CASE
END_METHOD

END_FUNCTION_BLOCK

// ---- POUs/Actuators/FB_CRYO_CMD_OVERRIDE.TcPOU
FUNCTION_BLOCK FB_CRYO_CMD_OVERRIDE
VAR_INPUT
	in_bEnable:		BOOL;			// External ON/OFF command.
	in_bCorrEngCmd:	BOOL := FALSE;	// Correct active ENG command when switching to MANUAL Mode.
END_VAR
VAR_OUTPUT
	out_bEnable:	BOOL := FALSE;	// Resulting command
	out_bError:		BOOL := FALSE;	// Error flag (bug in SW implementation)
	out_bInterlock:	BOOL := FALSE;	// Flag if any command is prevented
	out_bWarning:	BOOL := FALSE;	// ENG command set to a not permitted command
	out_sMode:		STRING := '';	// Active Mode
	out_sStatus:	STRING := 'OK';	// Textual description in case of problems
END_VAR
VAR
	bAutoMode:		BOOL := TRUE;	// AUTO=true, MANUAL=false
	bEngMode:		BOOL := FALSE;	// Commissioning/Engineering mode. Ignores interlocks
	
	
	// Disable/enable manual control buttons
	bDisableBtnOn:	BOOL := FALSE;
	bDisableBtnOff:	BOOL := FALSE;

	// ON/OFF command permissions
	bPermitOn:		BOOL := TRUE;
	bPermitOff:		BOOL := TRUE;
	
	// Manual command
	bManualCmd:		BOOL := FALSE;
	
	// Reset interlocks (if possible)
	bReset:			BOOL := FALSE;
END_VAR

// Interlock is active if any command is not allowed
out_bInterlock	:= (NOT bPermitOn) OR (NOT bPermitOff);

// Both commands cannot be prevented at the same time ==> error
out_bError	:= (NOT bPermitOn) AND (NOT bPermitOff);

// This should never happen. Indicates error in the implementation.
IF out_bError	THEN
	out_sStatus	:= 'ERROR: Both commands prevented!';
	RETURN;
ELSE
	out_sStatus	:= 'OK';
END_IF


IF bAutoMode THEN
	out_sMode	:= 'AUTO';
	
	// There are no warnings in AUTO mode.
	out_bWarning:= FALSE;
	
	// Disable Manual control buttons
	bDisableBtnOn	:= TRUE;
	bDisableBtnOff	:= TRUE;
	
	// Only permitted commands can be set. Otherwise, error.
	IF in_bEnable AND NOT bPermitOn THEN
		// Impossible condition ==> error
		out_sStatus	:= 'ERROR: System command TRUE not permitted!';
		out_bError	:= TRUE;
		RETURN;
	ELSIF NOT in_bEnable AND NOT bPermitOff THEN
		// Impossible condition ==> error
		out_sStatus	:= 'ERROR: System command FALSE not permitted!';
		out_bError	:= TRUE;
		RETURN;
	END_IF
	
	// IN command =+> OUT command.
	bManualCmd	:= in_bEnable;
	out_bEnable	:= in_bEnable;

ELSIF bEngMode	THEN
	out_sMode	:= 'ENG';
	
	// No restrictions, no safety !!!
	// User responsible for damage caused by wrong/dangerous commands.

	// Enable both buttons.
	bDisableBtnOn	:= FALSE;
	bDisableBtnOff	:= FALSE;
	
	// Only set a warning if the user selects a command that the system doesn't allow.
	IF bManualCmd AND NOT bPermitOn THEN
		out_sStatus	:= 'WARNING: Command TRUE is not safe!';
		out_bWarning:= TRUE;
	ELSIF NOT bManualCmd AND NOT bPermitOff THEN
		out_sStatus	:= 'WARNING: Command FALSE is not safe!';
		out_bWarning:= TRUE;
	ELSE
		out_sStatus	:= 'OK';
		out_bWarning:= FALSE;
	END_IF

	// Assign user command to the output without any checks !!!
	out_bEnable		:= bManualCmd;

ELSE	// Manual mode.
	out_sMode	:= 'MANUAL';
	
	// Enable only permitted buttons.
	bDisableBtnOn	:= NOT bPermitOn;
	bDisableBtnOff	:= NOT bPermitOff;
	
	IF in_bCorrEngCmd	THEN
		// When exiting ENG Mode, if this flag is set, 
		// correct command set in ENG Mode if not permitted.
		IF	bManualCmd = TRUE   AND  NOT bPermitOn  THEN
			bManualCmd	:= FALSE;	// Set command to OFF
		ELSIF	bManualCmd = FALSE   AND  NOT bPermitOff  THEN
			bManualCmd	:= TRUE;	// Set command to ON
		END_IF
	END_IF

	// Only set a warning if the user selects a command that the system doesn't allow.
	IF bManualCmd AND NOT bPermitOn THEN
		out_sStatus	:= 'WARNING: Command TRUE is not safe!';
		out_bWarning:= TRUE;
	ELSIF NOT bManualCmd AND NOT bPermitOff THEN
		out_sStatus	:= 'WARNING: Command FALSE is not safe!';
		out_bWarning:= TRUE;
	ELSE
		out_sStatus	:= 'OK';
		out_bWarning:= FALSE;
	END_IF

	// Set the output command
	out_bEnable		:= bManualCmd;
END_IF

METHOD M_SetAllPermitted
VAR_INPUT
END_VAR
bPermitOn	:= TRUE;
bPermitOff	:= TRUE;
END_METHOD

METHOD M_SetPermissionOff
VAR_INPUT
	in_bPermit:	BOOL;
END_VAR
bPermitOff	:= in_bPermit;
END_METHOD

METHOD M_SetPermissionOn
VAR_INPUT
	in_bPermit:	BOOL;
END_VAR
bPermitOn	:= in_bPermit;
END_METHOD

METHOD M_SetPermissions
VAR_INPUT
	in_bPermitOn:	BOOL;
	in_bPermitOff:	BOOL;
END_VAR
bPermitOn	:= in_bPermitOn;
bPermitOff	:= in_bPermitOff;
END_METHOD

END_FUNCTION_BLOCK

// ---- POUs/Utilities/FB_CRYO_THLD_BASE.TcPOU
FUNCTION_BLOCK FB_CRYO_THLD_BASE
VAR_INPUT
	in_nMode:		E_CRYO_THLD_MODE := E_CRYO_THLD_MODE.FIXED;
	in_aThld:		ARRAY [1..4] OF LREAL;	// Array of fixed thresholds. See E_CRYO_ALARM_LEVELS and E_CRYO_ALARM_IDX.
	in_aThldDelay:	ARRAY [1..4] OF UDINT;	// Array of delays for each threshold [ms].
	in_lrHyst:		LREAL := 0.0;			// Hysteresis value, percent or absolute (see in_bHystPct)
	in_bHystPct:	BOOL := TRUE;			// If TRUE, hysteresis is in %, otherwise absolute value.
	in_lrValue:		LREAL;					// Value to compare against the thresholds
	in_lrPar1:		LREAL := 0.0;			// Par1, e.g. temperature, for ACTIVE thresholds
END_VAR
VAR_OUTPUT
	out_aThld:			ARRAY [1..4] OF LREAL;	// Active thresholds
	out_nAlarmState:	E_CRYO_ALARM_LEVEL	:= E_CRYO_ALARM_LEVEL.NORMAL;	// Alarm state, e.g. ALARM_HIGH
	out_sAlarmState:	STRING := 'NORMAL';	// Alarm state as a string, e.g. 'ALARM HIGH'
END_VAR
VAR
	timer:	TON;
END_VAR

// Set thresholds
M_SetThresholds();

// Compare input value against the thresholds
M_CheckAlarms();

METHOD M_CheckAlarms : BOOL
VAR_INPUT
END_VAR
VAR
	lrHyst:	LREAL;
END_VAR

// Execute the delay timer.
timer();

//
// Check the input value against the thresholds
// and set alarms and warnings.
// If configured for, activate alarms after a delay.
// Note: the value is compared against the OUT Thresholds !!!
//
CASE out_nAlarmState OF
	E_CRYO_ALARM_LEVEL.NORMAL:
		IF in_lrValue > out_aThld[E_CRYO_ALARM_IDX.ALARM_HIGH] THEN
			IF in_aThldDelay[E_CRYO_ALARM_IDX.ALARM_HIGH] > 0	THEN
				// Activation delay is configured.
				// Start the timer and change state to WARNING_HIGH.
				timer(IN:=FALSE);
				timer(IN:=TRUE, PT:=UDINT_TO_TIME(in_aThldDelay[E_CRYO_ALARM_IDX.ALARM_HIGH]));
				out_nAlarmState	:= E_CRYO_ALARM_LEVEL.WARNING_HIGH;
			ELSE
				timer(IN:=FALSE);
				out_nAlarmState	:= E_CRYO_ALARM_LEVEL.ALARM_HIGH;
			END_IF
		ELSIF in_lrValue < out_aThld[E_CRYO_ALARM_IDX.ALARM_LOW] THEN
			IF in_aThldDelay[E_CRYO_ALARM_IDX.ALARM_LOW] > 0	THEN
				// Activation delay is configured.
				// Start the timer and change state to WARNING_LOW.
				timer(IN:=FALSE);
				timer(IN:=TRUE, PT:=UDINT_TO_TIME(in_aThldDelay[E_CRYO_ALARM_IDX.ALARM_LOW]));
				out_nAlarmState	:= E_CRYO_ALARM_LEVEL.WARNING_LOW;
			ELSE
				timer(IN:=FALSE);
				out_nAlarmState	:= E_CRYO_ALARM_LEVEL.ALARM_LOW;
			END_IF
		ELSIF in_lrValue > out_aThld[E_CRYO_ALARM_IDX.WARNING_HIGH] THEN
			IF in_aThldDelay[E_CRYO_ALARM_IDX.WARNING_HIGH] > 0	THEN
				// Activation delay is configured.
				// Activate the warning once the timer expires.
				timer(IN:=TRUE, PT:=UDINT_TO_TIME(in_aThldDelay[E_CRYO_ALARM_IDX.WARNING_HIGH]));
				IF timer.Q	THEN
					IF in_lrValue > out_aThld[E_CRYO_ALARM_IDX.ALARM_HIGH] THEN
						// It might be that due to the delay the alarm level has been reached.
						out_nAlarmState	:= E_CRYO_ALARM_LEVEL.ALARM_HIGH;
					ELSE
						out_nAlarmState	:= E_CRYO_ALARM_LEVEL.WARNING_HIGH;
					END_IF
				END_IF
			ELSE
				timer(IN:=FALSE);
				out_nAlarmState	:= E_CRYO_ALARM_LEVEL.WARNING_HIGH;
			END_IF
		ELSIF	in_lrValue < out_aThld[E_CRYO_ALARM_IDX.WARNING_LOW]	THEN
			IF in_aThldDelay[E_CRYO_ALARM_IDX.WARNING_LOW] > 0	THEN
				// Activation delay is configured.
				// Activate the warning once the timer expires.
				timer(IN:=TRUE, PT:=UDINT_TO_TIME(in_aThldDelay[E_CRYO_ALARM_IDX.WARNING_LOW]));
				IF timer.Q	THEN
					IF in_lrValue < out_aThld[E_CRYO_ALARM_IDX.ALARM_LOW] THEN
						// It might be that due to the delay the alarm level has been reached.
						out_nAlarmState	:= E_CRYO_ALARM_LEVEL.ALARM_LOW;
					ELSE
						out_nAlarmState	:= E_CRYO_ALARM_LEVEL.WARNING_LOW;
					END_IF
				END_IF
			ELSE
				timer(IN:=FALSE);
				out_nAlarmState	:= E_CRYO_ALARM_LEVEL.WARNING_LOW;
			END_IF
		ELSE
			timer(IN:=FALSE);
		END_IF
	E_CRYO_ALARM_LEVEL.WARNING_HIGH:
		lrHyst	:= M_GetHysteresis(E_CRYO_ALARM_IDX.WARNING_HIGH);
		IF	in_lrValue > out_aThld[E_CRYO_ALARM_IDX.ALARM_HIGH]	THEN
			IF in_aThldDelay[E_CRYO_ALARM_IDX.ALARM_HIGH] > 0	THEN
				// Activation delay is configured.
				// Activate the alarm once the timer expires.
				timer(IN:=TRUE, PT:=UDINT_TO_TIME(in_aThldDelay[E_CRYO_ALARM_IDX.ALARM_HIGH]));
				IF timer.Q	THEN
					out_nAlarmState	:= E_CRYO_ALARM_LEVEL.ALARM_HIGH;
				END_IF
			ELSE
				timer(IN:=FALSE);
				out_nAlarmState	:= E_CRYO_ALARM_LEVEL.ALARM_HIGH;
			END_IF
		ELSIF in_lrValue < (out_aThld[E_CRYO_ALARM_IDX.WARNING_HIGH] - lrHyst) THEN
			timer(IN:=FALSE);
			out_nAlarmState	:= E_CRYO_ALARM_LEVEL.NORMAL;
		ELSE
			timer(IN:=FALSE);
		END_IF
	E_CRYO_ALARM_LEVEL.WARNING_LOW:
		lrHyst	:= M_GetHysteresis(E_CRYO_ALARM_IDX.WARNING_LOW);
		IF	in_lrValue < out_aThld[E_CRYO_ALARM_IDX.ALARM_LOW]	THEN
			IF in_aThldDelay[E_CRYO_ALARM_IDX.ALARM_LOW] > 0	THEN
				// Activation delay is configured.
				// Activate the alarm once the timer expires.
				timer(IN:=TRUE, PT:=UDINT_TO_TIME(in_aThldDelay[E_CRYO_ALARM_IDX.ALARM_LOW]));
				IF timer.Q	THEN
					out_nAlarmState	:= E_CRYO_ALARM_LEVEL.ALARM_LOW;
				END_IF
			ELSE
				timer(IN:=FALSE);
				out_nAlarmState	:= E_CRYO_ALARM_LEVEL.ALARM_LOW;
			END_IF
		ELSIF in_lrValue > (out_aThld[E_CRYO_ALARM_IDX.WARNING_LOW] + lrHyst) THEN
			timer(IN:=FALSE);
			out_nAlarmState	:= E_CRYO_ALARM_LEVEL.NORMAL;
		ELSE
			timer(IN:=FALSE);
		END_IF
	E_CRYO_ALARM_LEVEL.ALARM_HIGH:
		lrHyst	:= M_GetHysteresis(E_CRYO_ALARM_IDX.ALARM_HIGH);
		IF in_lrValue < (out_aThld[E_CRYO_ALARM_IDX.ALARM_HIGH] - lrHyst) THEN
			out_nAlarmState	:= E_CRYO_ALARM_LEVEL.WARNING_HIGH;
		END_IF
	E_CRYO_ALARM_LEVEL.ALARM_LOW:
		lrHyst	:= M_GetHysteresis(E_CRYO_ALARM_IDX.ALARM_LOW);
		IF in_lrValue > (out_aThld[E_CRYO_ALARM_IDX.ALARM_LOW] + lrHyst) THEN
			out_nAlarmState	:= E_CRYO_ALARM_LEVEL.WARNING_LOW;
		END_IF
END_CASE

// Set alarm level labels
M_UserSetLabel(out_nAlarmState);
END_METHOD

METHOD M_GetHysteresis : LREAL
VAR_INPUT
	in_nIndex:	E_CRYO_ALARM_IDX;
END_VAR
VAR
	lrHyst:	LREAL;
END_VAR
//
// Get the absolute value of hysteresis.
// 
IF in_bHystPct THEN
	// The vaue is given as percentage of threshold.
	lrHyst	:= in_aThld[in_nIndex] * in_lrHyst / 100.0;
ELSE
	// The vaue is given as absolute value.
	lrHyst	:= in_lrHyst;
END_IF

M_GetHysteresis	:= ABS(lrHyst);
END_METHOD

METHOD M_SetThresholds : BOOL
VAR_INPUT
END_VAR
VAR
	i:	INT;
END_VAR
CASE in_nMode OF
	E_CRYO_THLD_MODE.FIXED:
		// Take the input array for thresholds
		FOR i:=1 TO 4 DO
			out_aThld[i]	:= in_aThld[i];
		END_FOR
	E_CRYO_THLD_MODE.ACTIVE:
		// Dynamically set thresholds
		M_UserSetActiveThresholds();
	E_CRYO_THLD_MODE.LAST_ACTIVE:
		// Keep last thresholds. Don't do anything.
		;
END_CASE
END_METHOD

METHOD M_UserSetActiveThresholds : BOOL
// This is a Dummy implementation of active thresholds.
// TODO User: Define specific implementation.
VAR_INPUT
END_VAR
VAR
	i:	INT;
END_VAR
// TODO User
// Define specific implementation.
// This is just an example.
//
out_aThld[E_CRYO_ALARM_IDX.ALARM_LOW]	:= in_aThld[E_CRYO_ALARM_IDX.ALARM_LOW]    + in_lrPar1;
out_aThld[E_CRYO_ALARM_IDX.WARNING_LOW]	:= in_aThld[E_CRYO_ALARM_IDX.WARNING_LOW]  + in_lrPar1;
out_aThld[E_CRYO_ALARM_IDX.WARNING_HIGH]	:= in_aThld[E_CRYO_ALARM_IDX.WARNING_HIGH] - in_lrPar1;
out_aThld[E_CRYO_ALARM_IDX.ALARM_HIGH]	:= in_aThld[E_CRYO_ALARM_IDX.ALARM_HIGH]   - in_lrPar1;
END_METHOD

METHOD M_UserSetLabel : BOOL
VAR_INPUT
	in_nLevel:	E_CRYO_ALARM_LEVEL;
END_VAR
//
// Set labels depending on the alarm level.
// This is the default implementation.
// To be overwritten by User if different labels are needed.
//
CASE in_nLevel OF
	E_CRYO_ALARM_LEVEL.ALARM_LOW:
		out_sAlarmState	:= 'ALARM LOW';
	E_CRYO_ALARM_LEVEL.WARNING_LOW:
		out_sAlarmState	:= 'WARNING LOW';
	E_CRYO_ALARM_LEVEL.NORMAL:
		out_sAlarmState	:= 'NORMAL';
	E_CRYO_ALARM_LEVEL.WARNING_HIGH:
		out_sAlarmState	:= 'WARNING HIGH';
	E_CRYO_ALARM_LEVEL.ALARM_HIGH:
		out_sAlarmState	:= 'ALARM HIGH';
END_CASE
END_METHOD

END_FUNCTION_BLOCK

// ---- POUs/Simulation/FB_CRYO_SIM_SINE.TcPOU
// Simulator that generates sine wave 
FUNCTION_BLOCK FB_CRYO_SIM_SINE
VAR_INPUT
	in_lrAmplitude:	LREAL := 1.0;
	in_nPeriod:		UDINT := 10000;
END_VAR
VAR_OUTPUT
	out_lrValue:	LREAL;
END_VAR
VAR
	
	{attribute 'OPC.UA.DA':='0'}
	timer:			TON;
	
	{attribute 'OPC.UA.DA':='0'}
	bInitialised:	BOOL := FALSE;		// Used to start timer for the first time
	
	{attribute 'OPC.UA.DA':='0'}
	i:	INT;

END_VAR
VAR_TEMP
	t1:	LREAL;
	t2:	LREAL;
	t3:	LREAL;
	t4:	LREAL;
END_VAR

// Check possible devision by zero
IF in_nPeriod = 0 THEN
	in_nPeriod	:= 1000;
END_IF

IF NOT bInitialised THEN
	bInitialised := TRUE;
	
	// Start timer for signal=FALSE
	timer(IN:=FALSE);
	timer(IN:=TRUE, PT:=UDINT_TO_TIME(in_nPeriod));
	RETURN;
END_IF

// Execute timer
// The timer is actually used just for the 'angle' for the sin().
// Angle = ET / PT * 2PI
timer();

// If the timer expired, just restart it
IF timer.Q THEN
		timer(IN:=FALSE);
		timer(IN:=TRUE, PT:=UDINT_TO_TIME(in_nPeriod));
END_IF

// Set the output
t1	:= TIME_TO_LREAL(timer.ET);
t2	:= TIME_TO_LREAL(timer.PT);
t3	:= t1 / t2 * 2 * 3.14;
t4	:= in_lrAmplitude * SIN(t3);

// Set output
out_lrValue	:= t4;

END_FUNCTION_BLOCK

// ---- POUs/Subsystems/Examples/Evacuation/FB_CRYO_EVAC_PDS.TcPOU
FUNCTION_BLOCK FB_CRYO_EVAC_PDS EXTENDS FB_CRYO_EVAC_BASE
VAR_INPUT
END_VAR
VAR_OUTPUT
END_VAR
VAR
	rp:	FB_CRYO_PUMP_MVP030;	// Roughing Pump
	tp:	FB_CRYO_PUMP_HIPACE30;	// Turbo Molecular Pump
	
END_VAR

SUPER^();

METHOD M_Configure
VAR_INPUT
END_VAR
//
// Specific PDS IR Imager configuration.
//
IF NOT stat.bConfigured	THEN
	// MANDATORY: Set References !!!
	// If not done, system will crash !!!
	rpRef	REF=rp;
	tpRef	REF=tp;
	

	// Specific instance configuration, e.g. anything different
	// from the default values given in the cfg structure of type T_CRYO_EVAC_CFG.
	cfg.nPressGaugeType1	:= E_CRYO_SENSOR_TYPE_PRESS.PKR_360;
	cfg.nPressGaugeType2	:= E_CRYO_SENSOR_TYPE_PRESS.PKR_360;

	cfg.lrThld_Prevac := 5.0;	// Prevacuum pressure threshold
	// Cryo pressure threshold to start Turbo Pump before opening Valve
	cfg.lrThld_TP_SafeStartPressure := 0.01;	
	// Cryo pressure threshold to start Turbo Pump once Valve is open
	cfg.lrThld_Valve_SafeOpenPressure := 0.1;	
	
	cfg.tDelay := T#3S;	// Time delay before stopping Turbo Pump

	stat.bConfigured	:= TRUE;;
ELSE
	RETURN;	// Nothing to do any more
END_IF
END_METHOD

METHOD M_ExecuteControllers
VAR_INPUT
END_VAR
//
// Specific PDS IR Imager HW.
//

// Roughing Pump	
rp(	
	in_bSimulation	:= FALSE,
	in_sName		:= 'MVP 030',
	in_bEnable		:= ctrl.bEnable_RP,
	in_nModel		:= 30,
	in_bAutoMonitor	:= TRUE,
	in_nPeriod		:= 3000);

// Turbo Molecular Pump
tp(	
	in_bSimulation	:= FALSE,
	in_sName		:= 'HIPACE 30',
	in_bEnable		:= ctrl.bEnable_TP,
	in_nModel		:= 30,
	in_bAutoMonitor	:= TRUE,
	in_nPeriod		:= 3000);


valve(in_bEnable	:= ctrl.bEnable_Valve);
END_METHOD

END_FUNCTION_BLOCK

// ---- POUs/Subsystems/Evacuation/FB_CRYO_EVAC_BASE.TcPOU
FUNCTION_BLOCK FB_CRYO_EVAC_BASE
VAR_INPUT
	in_bEnable:					BOOL := FALSE;	// System active while in_bEnable is TRUE
	in_lrCryoPressure:			LREAL;			// Cryo pressure
END_VAR
VAR_OUTPUT
END_VAR
VAR
	rpRef:	REFERENCE TO FB_CRYO_PUMP_BASE;		// Roughing Pump
	tpRef:	REFERENCE TO FB_CRYO_PUMP_BASE;		// Turbo Molecular Pump
	valve:	FB_CRYO_VALVE_CTRL;					// Insulation Valve
	
	press1:	FB_CRYO_SENSOR_PRESSURE;	// Prevacuum pressure gauge #1
	press2:	FB_CRYO_SENSOR_PRESSURE;	// Prevacuum pressure gauge #2
	prevac:	FB_CRYO_PRESSURE_VOTE;		// Prevacuum pressure 
	
	cfg:	T_CRYO_EVAC_CFG;
	ctrl:	T_CRYO_EVAC_CTRL;
	stat:	T_CRYO_EVAC_STAT;
	
	timer:	TON;
	trig:	R_TRIG;	// Start trigger
END_VAR

// NOTE: Configuration is set on the first cycle.
//       Once stat.bConfigured is TRUE, 
//       configuration is not updated any more.
M_Configure();

M_ReadSensors();

M_ExecuteControllers();

M_UpdateStatus();

M_StateMachine();

METHOD M_Activity_ClosingValve
VAR_INPUT
END_VAR
IF valve.stat.bActOFF THEN
	// The valve is closed.
	// Apply a delay before stopping Turbo pump.
	// Start the timer for the delay.
	timer(IN:=FALSE);
	timer(IN:=TRUE, PT:=cfg.tDelay);
	stat.nState	:= E_CRYO_EVAC_STATE.DELAY_STOPPING;	// Next state
	M_SetLabels();
END_IF
END_METHOD

METHOD M_Activity_DelayBeforeStoppingPumps
VAR_INPUT
END_VAR
timer();

IF timer.Q THEN
	// Delay timer expired.
	// Reset timer.
	timer(IN:=FALSE);
	
	// Stop Turbo Pump.
	ctrl.bEnable_TP	:= FALSE;
	stat.nState		:= E_CRYO_EVAC_STATE.STOP_T_PUMP;	// Next state
	M_SetLabels();
END_IF
END_METHOD

METHOD M_Activity_Evacuating
VAR_INPUT
END_VAR
// System is started by setting in_bEnable to TRUE
IF NOT in_bEnable THEN
	// If system is disabled, start stopping procedure.
	ctrl.bEnable_Valve	:= FALSE;
	stat.nState			:= E_CRYO_EVAC_STATE.CLOSE_INSULATION_VALVE;	// Next state
	M_SetLabels();
ELSIF prevac.stat.lrPressure > cfg.lrThld_Prevac THEN
	// Something is wrong. Prevacuum pressure is too high. Stop evacuation!
	// Set error
	M_SetError('Prevacuum pressure too high. Stopping evacuation...');
	ctrl.bEnable_Valve	:= FALSE;
	stat.nState			:= E_CRYO_EVAC_STATE.CLOSE_INSULATION_VALVE;	// Next state
	M_SetLabels();
END_IF
END_METHOD

METHOD M_Activity_Off
VAR_INPUT
END_VAR
// Disable anything that is not safe in this state
ctrl.bEnable_RP		:= FALSE;
ctrl.bEnable_TP		:= FALSE;
ctrl.bEnable_Valve	:= FALSE;


// System is started by setting in_bEnable to TRUE
trig(CLK := in_bEnable);

IF trig.Q THEN
	// Clear any existing error
	M_SetError('OK');
	
	// Enable Roughing Pump
	ctrl.bEnable_RP	:= TRUE;
	
	stat.nState	:= E_CRYO_EVAC_STATE.START_R_PUMP;	// Next state
	M_SetLabels();
END_IF
END_METHOD

METHOD M_Activity_OpeningValve
VAR_INPUT
END_VAR
IF NOT in_bEnable THEN
	// If system is disabled, start stopping procedure.
	ctrl.bEnable_Valve	:= FALSE;
	stat.nState			:= E_CRYO_EVAC_STATE.CLOSE_INSULATION_VALVE;	// Next state
	M_SetLabels();
ELSIF valve.stat.bActON THEN
	// The valve is open.
	// If valve was open before starting Turbo pump, 
	// wait for cryo pressure drop and then start the pump.
	// If the turbo pump is already running, the evacuation has started.
	IF NOT stat.bValveAfterTP	THEN
		stat.nState	:= E_CRYO_EVAC_STATE.WAIT_CRYO_VAC;	// Next state
	ELSE
		stat.nState	:= E_CRYO_EVAC_STATE.EVACUATING;	// Next state
	END_IF
	M_SetLabels();
END_IF
END_METHOD

METHOD M_Activity_StartingRoughingPump
VAR_INPUT
END_VAR
// Disable anything that is not safe in this state
ctrl.bEnable_TP		:= FALSE;
ctrl.bEnable_Valve	:= FALSE;


IF NOT in_bEnable THEN
	// If system is disabled, start stopping procedure.
	ctrl.bEnable_Valve	:= FALSE;
	stat.nState	:= E_CRYO_EVAC_STATE.CLOSE_INSULATION_VALVE;	// Next state
	M_SetLabels();
ELSIF rpRef.M_IsReady() THEN
	// Roughing Pump is Ready.
	// Wait for the prevacuum.
	stat.nState	:= E_CRYO_EVAC_STATE.WAIT_PREVAC;	// Next state
	M_SetLabels();
END_IF
END_METHOD

METHOD M_Activity_StartingTurboPump
VAR_INPUT
END_VAR
// Safety
// If the valve should be open after Turbo Pump has started,
// keep the valve closed.
IF stat.bValveAfterTP THEN
	ctrl.bEnable_Valve	:= FALSE;
END_IF

IF NOT in_bEnable THEN
	// If system is disabled, start stopping procedure.
	ctrl.bEnable_Valve	:= FALSE;
	stat.nState			:= E_CRYO_EVAC_STATE.CLOSE_INSULATION_VALVE;	// Next state
	M_SetLabels();
ELSIF tpRef.M_IsReady() THEN
	// Turbo Molecular Pump is Ready.
	// If the valve is not open, open it.
	// Otherwise, evacuation has started.
	IF stat.bValveAfterTP THEN
		ctrl.bEnable_Valve	:= TRUE;
		stat.nState			:= E_CRYO_EVAC_STATE.OPEN_INSULATION_VALVE;	// Next state
	ELSE
		stat.nState	:= E_CRYO_EVAC_STATE.EVACUATING;	// Next state
	END_IF
	M_SetLabels();
END_IF
END_METHOD

METHOD M_Activity_StoppingRoughingPump
VAR_INPUT
END_VAR
// Disable anything that is not safe in this state
ctrl.bEnable_RP		:= FALSE;
ctrl.bEnable_TP		:= FALSE;
ctrl.bEnable_Valve	:= FALSE;


// The evacuation system is in the process of shutting down.
// Allow re-starting of evacuation.
// System is started by setting in_bEnable to TRUE.
trig(CLK := in_bEnable);

IF trig.Q THEN
	// Clear any existing error
	M_SetError('OK');
	
	// Enable Roughing Pump
	ctrl.bEnable_RP	:= TRUE;
	
	stat.nState	:= E_CRYO_EVAC_STATE.START_R_PUMP;	// Next state
	M_SetLabels();
ELSIF NOT rpRef.M_IsRunning() THEN
	// The Roughing Pump stopped.
	// Wait for the Turbo Pump to get to complete stop.
	stat.nState	:= E_CRYO_EVAC_STATE.WAIT_T_PUMP_STOP;	// Next state
	M_SetLabels();
END_IF
END_METHOD

METHOD M_Activity_StoppingTurboPump
VAR_INPUT
END_VAR
// Disable anything that is not safe in this state
ctrl.bEnable_Valve	:= FALSE;


// The evacuation system is in the process of shutting down.
// Allow re-starting of evacuation.
// System is started by setting in_bEnable to TRUE.
trig(CLK := in_bEnable);

IF trig.Q THEN
	// Clear any existing error
	M_SetError('OK');
	
	// Enable Roughing Pump
	ctrl.bEnable_RP	:= TRUE;
	
	stat.nState	:= E_CRYO_EVAC_STATE.START_R_PUMP;	// Next state
	M_SetLabels();
ELSIF tpRef.M_GetSpeed() < 100 THEN
	// TODO: This is ATH2303M specific.
	//       Maybe, speed < 100 or similar check.
	
	// The Turbo Pump speed dropped below 100 rpm.
	// Stop the Roughing Pump.
	ctrl.bEnable_RP	:= FALSE;
	stat.nState		:= E_CRYO_EVAC_STATE.STOP_R_PUMP;	// Next state
	M_SetLabels();
END_IF
END_METHOD

METHOD M_Activity_WaitingCryoVacuum
VAR_INPUT
END_VAR
// Safety
// Disable Turbo Pump until it is safe to start.
ctrl.bEnable_TP	:= FALSE;

IF NOT in_bEnable THEN
	// If system is disabled, start stopping procedure.
	ctrl.bEnable_Valve	:= FALSE;
	stat.nState			:= E_CRYO_EVAC_STATE.CLOSE_INSULATION_VALVE;	// Next state
	M_SetLabels();
ELSIF in_lrCryoPressure <= cfg.lrThld_Valve_SafeOpenPressure THEN
	ctrl.bEnable_TP	:= TRUE;	// Enable Turbo Pump
	stat.nState		:= E_CRYO_EVAC_STATE.START_T_PUMP;	// Next state
	M_SetLabels();
END_IF
END_METHOD

METHOD M_Activity_WaitingPrevacuum
VAR_INPUT
END_VAR
// Disable anything that is not safe in this state
ctrl.bEnable_TP		:= FALSE;
ctrl.bEnable_Valve	:= FALSE;


IF NOT in_bEnable THEN
	// If system is disabled, start stopping procedure.
	ctrl.bEnable_Valve	:= FALSE;
	stat.nState	:= E_CRYO_EVAC_STATE.CLOSE_INSULATION_VALVE;	// Next state
	M_SetLabels();
ELSIF prevac.stat.lrPressure <= cfg.lrThld_Prevac THEN
	// If cryostat pressure is <= lrThldTP_SafeStartPressure, 
	// start Turbo Pump before opening the Insulation Valve.
	// Otherwise, open the Insulation Valve first.
	IF in_lrCryoPressure <= cfg.lrThld_TP_SafeStartPressure	THEN
		ctrl.bEnable_TP		:= TRUE;	// Enable Turbo Pump
		stat.bValveAfterTP	:= TRUE;	// Open valve after Turbo Pump has started
		stat.nState		:= E_CRYO_EVAC_STATE.START_T_PUMP;	// Next state
	ELSE
		ctrl.bEnable_Valve	:= TRUE;	// Open Valve
		stat.bValveAfterTP	:= FALSE;	// Valve opens before Turbo Pump starts
		stat.nState			:= E_CRYO_EVAC_STATE.OPEN_INSULATION_VALVE;	// Next state
	END_IF
	M_SetLabels();
END_IF
END_METHOD

METHOD M_Activity_WaitingTurboPump2Stop
VAR_INPUT
END_VAR
// Disable anything that is not safe in this state
ctrl.bEnable_RP		:= FALSE;
ctrl.bEnable_TP		:= FALSE;
ctrl.bEnable_Valve	:= FALSE;


// The evacuation system is in the process of shutting down.
// Allow re-starting of evacuation.
// System is started by setting in_bEnable to TRUE.
trig(CLK := in_bEnable);

IF trig.Q THEN
	// Clear any existing error
	M_SetError('OK');
	
	// Enable Roughing Pump
	ctrl.bEnable_RP	:= TRUE;
	
	stat.nState	:= E_CRYO_EVAC_STATE.START_R_PUMP;	// Next state
	M_SetLabels();
ELSIF tpRef.M_GetSpeed() = 0 THEN
	// The Turbo Pump came to complete stop.
	// The Evacuation system is OFF.
	stat.nState	:= E_CRYO_EVAC_STATE.OFF;	// Next state
	M_SetLabels();
END_IF
END_METHOD

METHOD M_Configure
VAR_INPUT
END_VAR
//
// TODO USER: If needed, overload this method with specific values.
//            This is the default configuration.
//
IF NOT stat.bConfigured	THEN
	// Specific instance configuration, e.g. anything different
	// from the default values given in the cfg structure of type T_CRYO_EVAC_CFG.
	cfg.nPressGaugeType1	:= E_CRYO_SENSOR_TYPE_PRESS.PKR_360;
	cfg.nPressGaugeType2	:= E_CRYO_SENSOR_TYPE_PRESS.PKR_360;

	cfg.lrThld_Prevac := 5.0;	// Prevacuum pressure threshold 5 mbar
	// Cryo pressure threshold to start Turbo Pump before opening Valve 10e-2 mbar
	cfg.lrThld_TP_SafeStartPressure := 0.01;	 
	// Cryo pressure threshold to start Turbo Pump once Valve is open 10e-1 mbar
	cfg.lrThld_Valve_SafeOpenPressure := 0.1;	
	cfg.tDelay := T#3S;	// Time delay before stopping Turbo Pump

	stat.bConfigured	:= TRUE;;
ELSE
	RETURN;	// Nothing to do any more
END_IF
END_METHOD

METHOD M_ExecuteControllers
VAR_INPUT
END_VAR
END_METHOD

METHOD M_GotoOff
VAR_INPUT
END_VAR
ctrl.bEnable_TP		:= FALSE;
ctrl.bEnable_RP		:= FALSE;
ctrl.bEnable_Valve	:= FALSE;
stat.nState			:= E_CRYO_EVAC_STATE.OFF;	// Next state
M_SetLabels();
END_METHOD

METHOD M_ReadSensors
VAR_INPUT
END_VAR
// Read prevacuum pressure sensors.
// Note: Pressure sensor type is configured in cfg.
//       Default is Pfeiffer PKR 360 KF25.
press1(in_nType := cfg.nPressGaugeType1, in_nSampleTime := 100);
press2(in_nType := cfg.nPressGaugeType2, in_nSampleTime := 100);
prevac(
	in_bSimulation	:= cfg.bPressSimulation,
	in_nNumSensor	:= 2,
	in_nVoteMethod	:= E_CRYO_VOTE.V_1oo2,
	in_pSensor1		:= ADR(press1),
	in_pSensor2		:= ADR(press2));
END_METHOD

METHOD M_SetError
VAR_INPUT
	in_sErrorText:	STRING(64);
END_VAR
stat.bError		:= (in_sErrorText <> 'OK');
stat.sErrorText	:= in_sErrorText;
END_METHOD

METHOD M_SetLabels
VAR_INPUT
END_VAR
VAR
    fbFormat:	FB_FormatString;
	nVal:		UDINT;
	lrVal:		LREAL;
END_VAR
CASE stat.nState	OF
	E_CRYO_EVAC_STATE.NONE:
		stat.sState		:= 'NONE';
		stat.sStatus	:= 'UNKNOWN';
	E_CRYO_EVAC_STATE.OFF:
		stat.sState		:= 'OFF';
		stat.sStatus	:= 'OFF';
	E_CRYO_EVAC_STATE.START_R_PUMP:
		stat.sState		:= 'START_R_PUMP';
		stat.sStatus	:= 'Starting Roughing Pump...';
	E_CRYO_EVAC_STATE.WAIT_PREVAC:
		stat.sState		:= 'WAIT_PREVAC';
		fbFormat(	sFormat := 'Waiting Prevacuum Pressure <= %.4f [mbar]...', 
					arg1 := F_LREAL(cfg.lrThld_Prevac), 
					sOut => stat.sStatus);
	E_CRYO_EVAC_STATE.OPEN_INSULATION_VALVE:
		stat.sState		:= 'OPEN_INSULATION_VALVE';
		stat.sStatus	:= 'Opening Insulation Valve...';
	E_CRYO_EVAC_STATE.START_T_PUMP:
		stat.sState		:= 'START_T_PUMP';
		stat.sStatus	:= 'Starting Turbo Molecular Pump...';
	E_CRYO_EVAC_STATE.WAIT_CRYO_VAC:
		stat.sState		:= 'WAIT_CRYO_VAC';
		// The target cryostat pressure depends on whether the valve is open or not.
		IF valve.stat.bActON THEN
			lrVal	:= cfg.lrThld_Valve_SafeOpenPressure;
		ELSE
			lrVal	:= cfg.lrThld_TP_SafeStartPressure;
		END_IF
		fbFormat(	sFormat := 'Waiting Cryostat Pressure <= %.4f [mbar]...', 
					arg1 := F_LREAL(lrVal), 
					sOut => stat.sStatus);
	E_CRYO_EVAC_STATE.EVACUATING:
		stat.sState		:= 'EVACUATING';
		stat.sStatus	:= 'EVACUATING...';
	E_CRYO_EVAC_STATE.CLOSE_INSULATION_VALVE:
		stat.sState		:= 'CLOSE_INSULATION_VALVE';
		stat.sStatus	:= 'Closing Insulation Valve...';
	E_CRYO_EVAC_STATE.DELAY_STOPPING:
		stat.sState		:= 'DELAY_STOPPING';
		nVal			:= TIME_TO_UDINT(cfg.tDelay);
		fbFormat(	sFormat := 'Delay of %d [ms] Before Stopping Pumps...', 
					arg1 := F_UDINT(nVal), 
					sOut => stat.sStatus);
	E_CRYO_EVAC_STATE.STOP_T_PUMP:
		stat.sState		:= 'STOP_T_PUMP';
		stat.sStatus	:= 'Stopping Turbo Molecular Pump...';
	E_CRYO_EVAC_STATE.STOP_R_PUMP:
		stat.sState		:= 'STOP_R_PUMP';
		stat.sStatus	:= 'Stopping Roughing Pump...';
	E_CRYO_EVAC_STATE.WAIT_T_PUMP_STOP:
		stat.sState		:= 'WAIT_T_PUMP_STOP';
		stat.sStatus	:= 'Waiting for Turbo Molecular Pump to Stop...';
	
END_CASE
END_METHOD

METHOD M_StateMachine
VAR_INPUT
END_VAR
CASE stat.nState	OF
	E_CRYO_EVAC_STATE.NONE:
		M_GotoOff();
	E_CRYO_EVAC_STATE.OFF:
		M_Activity_Off();
	E_CRYO_EVAC_STATE.START_R_PUMP:
		M_Activity_StartingRoughingPump();
	E_CRYO_EVAC_STATE.WAIT_PREVAC:
		M_Activity_WaitingPrevacuum();
	E_CRYO_EVAC_STATE.OPEN_INSULATION_VALVE:
		M_Activity_OpeningValve();
	E_CRYO_EVAC_STATE.START_T_PUMP:
		M_Activity_StartingTurboPump();
	E_CRYO_EVAC_STATE.WAIT_CRYO_VAC:
		M_Activity_WaitingCryoVacuum();
	E_CRYO_EVAC_STATE.EVACUATING:
		M_Activity_Evacuating();
	E_CRYO_EVAC_STATE.CLOSE_INSULATION_VALVE:
		M_Activity_ClosingValve();
	E_CRYO_EVAC_STATE.DELAY_STOPPING:
		M_Activity_DelayBeforeStoppingPumps();
	E_CRYO_EVAC_STATE.STOP_T_PUMP:
		M_Activity_StoppingTurboPump();
	E_CRYO_EVAC_STATE.STOP_R_PUMP:
		M_Activity_StoppingRoughingPump();
	E_CRYO_EVAC_STATE.WAIT_T_PUMP_STOP:
		M_Activity_WaitingTurboPump2Stop();
	
END_CASE
END_METHOD

METHOD M_UpdateStatus
VAR_INPUT
END_VAR
stat.bEnabled		:= in_bEnable;
stat.bRootPumpON	:= rpRef.M_IsReady();
stat.bTurboPumpON	:= tpRef.M_IsReady();
stat.bValveOpen		:= valve.stat.bActON;
END_METHOD

END_FUNCTION_BLOCK

// ---- POUs/Pumps/FB_CRYO_PUMP_BASE.TcPOU
// Cryo Pump Control Base FB
FUNCTION_BLOCK FB_CRYO_PUMP_BASE EXTENDS FB_RS_BASE
VAR_INPUT
	{attribute 'OPC.UA.DA' := '0'}
	in_bEnable:			BOOL;			// Flag to Start/Stop pump
	{attribute 'OPC.UA.DA' := '0'}
	in_nModel:			DINT := 2303;	// Model number
	{attribute 'OPC.UA.DA' := '0'}
	in_bAutoMonitor:	BOOL := TRUE;	// If true, it starts PERIODIC reads (monitoring) after INIT
	{attribute 'OPC.UA.DA' := '0'}
	in_nPeriod:			DINT := 10000;	// Interval for periodic reading [ms], default 10000 ms = 10 sec
END_VAR
VAR_OUTPUT
END_VAR
VAR
	{attribute 'OPC.UA.DA' := '0'}
	cfgBaseRef:			REFERENCE TO T_CRYO_PUMP_BASE_CFG;	
	{attribute 'OPC.UA.DA' := '0'}
	ctrlBaseRef:		REFERENCE TO T_CRYO_PUMP_BASE_CTRL;	
	{attribute 'OPC.UA.DA' := '0'}
	statBaseRef:		REFERENCE TO T_CRYO_PUMP_BASE_STAT;	

	// Pointers to arrays of INIT and READ commands
	{attribute 'OPC.UA.DA' := '0'}
	ptrInitCmds:	POINTER TO ARRAY [1..8]  OF T_CRYO_PUMP_CMD;(* Pointer to INIT commands *)
	{attribute 'OPC.UA.DA' := '0'}
	ptrReadCmds:	POINTER TO ARRAY [1..16] OF T_CRYO_PUMP_CMD;(* Pointer to READ commands *)


	(* Timers *)
	{attribute 'OPC.UA.DA' := '0'}
	fbTimer:		TON; 	// General Timeout
	timerState:		TON;	// Timer for state changes
	
	// Triggers
	triggerStart:	R_TRIG;
	triggerStop:	F_TRIG;
	

	(* Misc internal vars *)
	{attribute 'OPC.UA.DA' := '0'}
	cmdCounter:		INT := 1;	// Position in commands table
	{attribute 'OPC.UA.DA' := '0'}
	bResult:		BOOL := FALSE;
	{attribute 'OPC.UA.DA' := '0'}
	bStarted:		BOOL := FALSE;

	// TODO: Add Input signals in Fbs that EXTEND this FB.

	// Output signals
	q_bStart		AT %Q*:	BOOL;	// Start/Stop the pump. Common to all.

END_VAR

// Hard-coded configuration
M_Configure();

(* Execute comm instance *)
M_ExecuteComm();
//comm(in_sCmdSuffix:=in_sCmdSuffix, in_sReplySuffix:=in_sReplySuffix, in_nTimeout:=3000);

// Update pump status from digital signals.
M_UpdateStatus();

// Capture Start/Stop commands and execute the State Machine
M_StateMachine();

// Execute the base class object FB_RS_BASE
SUPER^();

METHOD ActivityInitializing
VAR_INPUT
	bExecute:	BOOL;
END_VAR
VAR_INST
	{attribute 'OPC.UA.DA' := '0'}
    nMethodState:	INT := 0;	// State Machine current state
END_VAR
END_METHOD

METHOD ActivityMonitoring
VAR_INPUT
	bExecute:	BOOL;
END_VAR
VAR_INST
	{attribute 'OPC.UA.DA' := '0'}
    nMethodState:	INT := 0;	// State Machine current state
	{attribute 'OPC.UA.DA' := '0'}
	nRetries:		INT := 0;	// Number of retries in case of communication problems
END_VAR

VAR
	offset: INT;
END_VAR
END_METHOD

METHOD CheckForEvents
VAR_INPUT
END_VAR
VAR
END_VAR

(* 
	Start assuming the HW is OK in case there was no communication problem. 
	This is needed to recover from the situation where 
	the HW was failing and now it is working.
*)

//IF NOT bCommProblem	THEN
//	nInternalEvent := E_SM_EVENT.HWOK;
//END_IF




(* 
	Check for events in the following order: 
   	1) HW failure: without HW avilability there is no point to do anything
	2) Internal events: to allow completing the initiated commands before 
                        starting processing new commands. 
   	3) Commands: to react to external commands. Commands should be executed 
                 before processing HW signals to allow to start a recovery action.
   	4) HW signals: if any.
*)

IF NOT M_GetCouplerState() THEN	
	(* Check if the HW is NOT OK *)
	(*
	If the hardware status is NOT OK, we cannot trust the readings.
	Variable i_nCouplerState has to be mapped to a State of a terminal, e.g. EK1100.
	The value should be 8.
 	*)
	SetEvent(E_SM_EVENT.ERRHW);
	SetStatus(E_SM_ERROR.HW_NOT_OP, 'ERROR: HW not in OPERATIONAL state');
	
ELSIF M_GetCouplerState() AND statRef.nErrorCode = E_SM_ERROR.HW_NOT_OP THEN
	SetEvent(E_SM_EVENT.HWOK);

ELSIF ctrlRef.bExecute  THEN
	(* Handle commands *)
	ctrlRef.bExecute		:= FALSE;			(* Clear the Execute bit *)
	SetLastCommand(ctrlRef.nCommand);			(* Save the last command *)
	SetEvent(ctrlRef.nCommand);
	ctrlRef.nCommand 	:= E_RS_COMMAND.NONE;	(* Clear the Command *)
ELSIF nInternalEvent <> E_SM_EVENT.NONE THEN
	(* Handle internal events *)
	SetEvent(nInternalEvent);
	nInternalEvent := E_SM_EVENT.NONE;
ELSE
	(* Handle HW problems and unexpected bahaviour *)
	
END_IF
END_METHOD

METHOD M_Configure
VAR_INPUT
END_VAR
VAR
	
END_VAR
// TODO: Implement specific configuration
END_METHOD

METHOD M_ExecuteComm
VAR_INPUT
END_VAR
END_METHOD

METHOD M_GetCouplerState : BOOL
VAR_INPUT
END_VAR
END_METHOD

METHOD M_GetSpeed : DINT
VAR_INPUT
END_VAR
END_METHOD

METHOD M_IsReady : BOOL
VAR_INPUT
END_VAR
END_METHOD

METHOD M_IsRunning : BOOL
VAR_INPUT
END_VAR
END_METHOD

METHOD M_StateMachine
VAR_INPUT
END_VAR
//////////////////////
// Pump State Machine
//////////////////////
CASE statBaseRef.nPumpState OF
	E_CRYO_PUMP_STATE.OFF:
		// Capture START command
		triggerStart(CLK:=in_bEnable);
		IF triggerStart.Q THEN
			// in_bEnable is TRUE, start the pump.
			ctrlBaseRef.bStart		:= TRUE;
			statBaseRef.nPumpState	:= 	E_CRYO_PUMP_STATE.STARTING;
			statBaseRef.sPumpState	:= 'Starting...';
			// Restart the timer
			timerState(IN:=FALSE);
			timerState(IN:=TRUE,PT:=UDINT_TO_TIME(cfgBaseRef.nTimeoutState));
		END_IF
	E_CRYO_PUMP_STATE.STARTING:
		timerState();
		triggerStop(CLK:= in_bEnable);
		IF timerState.Q THEN
			// Timeout, stop the pump.
			ctrlBaseRef.bStart		:= FALSE;
			timerState(IN:=FALSE);
			statBaseRef.nPumpState	:= 	E_CRYO_PUMP_STATE.ERROR;
			statBaseRef.sPumpState	:= 'ERROR - Timeout on START';
		ELSIF M_IsReady() THEN
			timerState(IN:=FALSE);
			statBaseRef.nPumpState	:= 	E_CRYO_PUMP_STATE.ON;
			statBaseRef.sPumpState	:= 'ON';
		ELSIF triggerStop.Q THEN
			// in_bEnable is FALSE, stop the pump.
			ctrlBaseRef.bStart		:= FALSE;
			// Restart the timer
			timerState(IN:=FALSE);
			timerState(IN:=TRUE,PT:=UDINT_TO_TIME(cfgBaseRef.nTimeoutState));
			statBaseRef.nPumpState	:= 	E_CRYO_PUMP_STATE.STOPPING;
			statBaseRef.sPumpState	:= 'Stopping...';
		END_IF
	E_CRYO_PUMP_STATE.ON:
		triggerStop(CLK:= in_bEnable);
		IF triggerStop.Q THEN
			// in_bEnable is FALSE, stop the pump.
			// Restart the timer
			ctrlBaseRef.bStart		:= FALSE;
			timerState(IN:=FALSE);
			timerState(IN:=TRUE,PT:=UDINT_TO_TIME(cfgBaseRef.nTimeoutState));
			statBaseRef.nPumpState	:= 	E_CRYO_PUMP_STATE.STOPPING;
			statBaseRef.sPumpState	:= 'Stopping...';
		ELSIF NOT M_IsReady()  OR  NOT M_IsRunning() THEN
			ctrlBaseRef.bStart		:= FALSE;
			statBaseRef.nPumpState	:= 	E_CRYO_PUMP_STATE.ERROR;
			statBaseRef.sPumpState	:= 'ERROR - Unexpected STOP';
		END_IF
	E_CRYO_PUMP_STATE.STOPPING:
		timerState();
		// Capture START command
		triggerStart(CLK:=in_bEnable);
		IF timerState.Q THEN
			timerState(IN:=FALSE);
			statBaseRef.nPumpState	:= 	E_CRYO_PUMP_STATE.ERROR;
			statBaseRef.sPumpState	:= 'ERROR - Timeout on STOP';
		ELSIF NOT M_IsReady()  AND NOT M_IsRunning() THEN
			timerState(IN:=FALSE);
			statBaseRef.nPumpState	:= 	E_CRYO_PUMP_STATE.OFF;
			statBaseRef.sPumpState	:= 'OFF';
		ELSIF triggerStart.Q THEN
			// in_bEnable is TRUE, start the pump.
			ctrlBaseRef.bStart		:= TRUE;
			statBaseRef.nPumpState	:= 	E_CRYO_PUMP_STATE.STARTING;
			statBaseRef.sPumpState	:= 'Starting...';
			// Restart the timer
			timerState(IN:=FALSE);
			timerState(IN:=TRUE,PT:=UDINT_TO_TIME(cfgBaseRef.nTimeoutState));
		END_IF
	E_CRYO_PUMP_STATE.ERROR:
		// To recover from error, STOP command has to be issued
		// in order to reset triggerStop.
		// Capture STOP command
		triggerStop(CLK:=in_bEnable);
		IF triggerStop.Q THEN
			// in_bEnable is TRUE, start the pump.
			statBaseRef.nPumpState	:= 	E_CRYO_PUMP_STATE.OFF;
			statBaseRef.sPumpState	:= 'OFF';
		END_IF
		
		// If in_bEnable is FALSE, Capture START command.
		triggerStart(CLK:=in_bEnable);
		IF triggerStart.Q THEN
			// in_bEnable is TRUE, start the pump.
			ctrlBaseRef.bStart		:= TRUE;
			statBaseRef.nPumpState	:= 	E_CRYO_PUMP_STATE.STARTING;
			statBaseRef.sPumpState	:= 'Starting...';
			// Restart the timer
			timerState(IN:=FALSE);
			timerState(IN:=TRUE,PT:=UDINT_TO_TIME(cfgBaseRef.nTimeoutState));
		END_IF
END_CASE


// Update outputs
q_bStart	:= ctrlBaseRef.bStart;
END_METHOD

METHOD M_UpdateStatus
VAR_INPUT
END_VAR
// TODO: For each pump FB that extends FB_CRYO_PUMP_BASE update inputs in M_UpdateStatus(), e.g.

(*
// Update inputs
stat.bReady		:= i_bReady;
stat.bSpeed100	:= i_bSpeed100;
stat.bWarning	:= i_bWarning;
stat.bAlarm		:= i_bAlarm;

CASE stat.nCtrlMode	OF
	0:	stat.sCtrlMode	:= 'HHR (Hand-Held Remote)';
	1:	stat.sCtrlMode	:= 'REMOTE';
	2:	stat.sCtrlMode	:= 'SERIAL LINK';
	3:	stat.sCtrlMode	:= 'FIELDBUS';
ELSE
	stat.sCtrlMode	:= 'UNKNOWN';
END_CASE

*)
END_METHOD

METHOD ProcessEvents
VAR_INPUT
END_VAR

(* 
	Before processing the event, execute the Do-Activity tasks. 
	Note that, in case of orthogonal regions, more than one Do-Activity 
	could run in the same PLC cycle.
	Note: Most of these activities have timeouts since they take time.
*)

IF	statRef.nSubstate = E_RS_BASE_SUBSTATE.OP_MONITORING 		OR 
	statRef.nSubstate = E_RS_BASE_SUBSTATE.NOTOP_READY			OR
	(statRef.nSubstate = E_RS_BASE_SUBSTATE.NOTOP_ERROR 	AND 
	 nLastGoodSubstate = E_RS_BASE_SUBSTATE.NOTOP_READY) 		OR 
	(statRef.nSubstate = E_RS_BASE_SUBSTATE.OP_ERROR 		AND 
	 nLastGoodSubstate = E_RS_BASE_SUBSTATE.OP_MONITORING)			THEN
	ActivityMonitoring(TRUE);
ELSIF statRef.nSubstate = E_RS_BASE_SUBSTATE.OP_MONITORING_USER THEN
	ActivityMonitoringUser(TRUE);
ELSIF statRef.nSubstate = E_RS_BASE_SUBSTATE.NOTOP_INITIALIZING THEN
	ActivityInitializing(TRUE);
END_IF

// Set last known good substate. Used for recovery from comm problems.
M_SetLastGoodSubstate();

(* 
	Evaluate state machine transitions.
*)

CASE statRef.nState OF

//***********************************
// NOTOP
//***********************************
E_RS_BASE_STATE.NOTOP:

	(* Transitions from NOTOP substates *)
	CASE statRef.nSubstate OF
	
	E_RS_BASE_SUBSTATE.NOTOP_NOTREADY:		
		IF 	nEvent = E_SM_EVENT.INIT OR cfgRef.bAutoMonitor  THEN
			nEvent := E_SM_EVENT.INIT;
			ActionInitExecute();
			SetState(E_RS_BASE_STATE.NOTOP, E_RS_BASE_SUBSTATE.NOTOP_INITIALIZING);
			SetStatus(E_SM_ERROR.OK, 'OK');
			RETURN;
		END_IF
		
	E_RS_BASE_SUBSTATE.NOTOP_INITIALIZING:			
		IF nEvent = E_SM_EVENT.INITDONE THEN
			nReadType := E_RS_BASE_READ_TYPE.PERIODIC;
			ActivityMonitoring(FALSE);	// Reset Monitoring method
			IF cfgRef.bAutoMonitor THEN
				nEvent := E_SM_EVENT.ENABLE;
				statRef.bAutoStarted	:= TRUE;
				SetState(E_RS_BASE_STATE.OP, E_RS_BASE_SUBSTATE.OP_MONITORING);
			ELSE
				SetState(E_RS_BASE_STATE.NOTOP, E_RS_BASE_SUBSTATE.NOTOP_READY);
			END_IF
			RETURN;
		ELSIF nEvent = E_SM_EVENT.ERRINIT THEN
			// INIT failed. Keep re-trying.
			SetState(E_RS_BASE_STATE.NOTOP, E_RS_BASE_SUBSTATE.NOTOP_NOTREADY);
			RETURN;
		END_IF
		
	E_RS_BASE_SUBSTATE.NOTOP_READY:			
		IF nEvent = E_SM_EVENT.ENABLE THEN
			IF cfgRef.bAutoMonitor THEN
				// Monitoring is already in progress.
				// It has to complete the read cycle in a clean way.
				nNextState		:= E_RS_BASE_STATE.OP;					// Next state after STOP	
				nNextSubstate	:= E_RS_BASE_SUBSTATE.OP_MONITORING;	// Next substate after STOP	
				nNextDescription:= 'BUSY';
				nReadType		:= E_RS_BASE_READ_TYPE.PERIODIC;
				RETURN;
			ELSE
				SetState(E_RS_BASE_STATE.OP, E_RS_BASE_SUBSTATE.OP_MONITORING);
				// This call MUST be after SetState()
				ActivityMonitoring(FALSE);	// Reset Monitoring method
			END_IF
		END_IF

	E_RS_BASE_SUBSTATE.NOTOP_ERROR:			
		IF nEvent = E_SM_EVENT.HWOK THEN
			SetState(E_RS_BASE_STATE.NOTOP, E_RS_BASE_SUBSTATE.NOTOP_NOTREADY);
			RETURN;
		ELSIF nEvent = E_SM_EVENT.COMMOK THEN
			SetState(E_RS_BASE_STATE.NOTOP, nLastGoodSubstate);
			RETURN;			
		END_IF
		
	END_CASE

	(* Transitions from NOTOP state *)
	IF	nEvent = E_SM_EVENT.ERRHW OR
		nEvent = E_SM_EVENT.ERRCOMM	THEN
		ActionUnexpExecute();
		SetState(E_RS_BASE_STATE.NOTOP, E_RS_BASE_SUBSTATE.NOTOP_ERROR);
		RETURN;
	END_IF
	
//***********************************
// OPERATIONAL
//***********************************
E_RS_BASE_STATE.OP:

	(* Transitions from OP subastates *)
	CASE statRef.nSubstate OF
	E_RS_BASE_SUBSTATE.OP_ERROR:			
		IF nEvent = E_SM_EVENT.HWOK THEN
			SetStatus(E_SM_ERROR.OK, 'OK');
			SetState(E_RS_BASE_STATE.OP, E_RS_BASE_SUBSTATE.OP_IDLE);
			RETURN;			
		ELSIF nEvent = E_SM_EVENT.DISABLE THEN
			ActionDisableExecute();
			SetState(E_RS_BASE_STATE.NOTOP, E_RS_BASE_SUBSTATE.NOTOP_ERROR);
			RETURN;			
		ELSIF nEvent = E_SM_EVENT.COMMOK THEN
			SetState(E_RS_BASE_STATE.OP, nLastGoodSubstate);
			RETURN;			
		END_IF

	E_RS_BASE_SUBSTATE.OP_MONITORING:
		IF nEvent = E_SM_EVENT.DISABLE THEN
			ActionDisableExecute();
			RETURN;			
		ELSIF nEvent = E_SM_EVENT.STOPMON THEN
			ActionStopExecute();
			RETURN;			
		ELSIF nEvent = E_SM_EVENT.READDONE THEN
			SetState(E_RS_BASE_STATE.OP, E_RS_BASE_SUBSTATE.OP_IDLE);
			RETURN;			
		ELSIF nEvent = E_SM_EVENT.ERRCOMM THEN
			SetState(E_RS_BASE_STATE.OP, E_RS_BASE_SUBSTATE.OP_ERROR);
			RETURN;			
		END_IF
		
	E_RS_BASE_SUBSTATE.OP_MONITORING_USER:			
		IF nEvent = E_SM_EVENT.DISABLE THEN
			ActionDisableExecute();
			RETURN;			
		ELSIF nEvent = E_SM_EVENT.STOPMON THEN
			ActionStopExecute();
			RETURN;			
		ELSIF nEvent = E_SM_EVENT.READDONE THEN
			SetState(E_RS_BASE_STATE.OP, E_RS_BASE_SUBSTATE.OP_IDLE);
			RETURN;			
		END_IF
		
	E_RS_BASE_SUBSTATE.OP_IDLE:			
		IF nEvent = E_SM_EVENT.DISABLE THEN
			ActionDisableExecute();
			RETURN;			
		ELSIF nEvent = E_SM_EVENT.READ THEN
			nReadType	:= E_RS_BASE_READ_TYPE.SINGLE;
			ActivityMonitoring(FALSE);	// Reset Monitoring method
			SetState(E_RS_BASE_STATE.OP, E_RS_BASE_SUBSTATE.OP_MONITORING);
			RETURN;			
		ELSIF nEvent = E_SM_EVENT.READ_USER THEN
			nReadType	:= E_RS_BASE_READ_TYPE.SINGLE_USER;
			ActivityMonitoringUser(FALSE);	// Reset Monitoring method
			SetState(E_RS_BASE_STATE.OP, E_RS_BASE_SUBSTATE.OP_MONITORING_USER);
			RETURN;			
		ELSIF nEvent = E_SM_EVENT.MONITOR OR nEvent = E_SM_EVENT.ENABLE THEN
			nReadType	:= E_RS_BASE_READ_TYPE.PERIODIC;
			ActivityMonitoring(FALSE);	// Reset Monitoring method
			SetState(E_RS_BASE_STATE.OP, E_RS_BASE_SUBSTATE.OP_MONITORING);
			RETURN;			
		ELSIF nEvent = E_SM_EVENT.MONITOR_USER THEN
			nReadType	:= E_RS_BASE_READ_TYPE.PERIODIC_USER;
			ActivityMonitoringUser(FALSE);	// Reset Monitoring method
			SetState(E_RS_BASE_STATE.OP, E_RS_BASE_SUBSTATE.OP_MONITORING_USER);
			RETURN;			
		END_IF
		
	END_CASE
	
	// Transitions from OP state.
	// Valid for any OP substate.
	IF nEvent = E_SM_EVENT.ERRHW THEN
		ActionUnexpExecute();
		SetState(E_RS_BASE_STATE.OP, E_RS_BASE_SUBSTATE.OP_ERROR);
		RETURN;
	ELSIF nEvent = E_SM_EVENT.ERRCOMM THEN
		SetState(E_RS_BASE_STATE.OP, E_RS_BASE_SUBSTATE.OP_ERROR);
		RETURN;
	END_IF
	
END_CASE

(* 
	"Global" internal transitions valid in any state should go here.
	They do not change the active state configuration. 
	They are evaluated after all the others transitions have been 
	considered.
*) 
IF nEvent = E_SM_EVENT.RESET THEN
	ActionResetExecute();
	SetState(E_RS_BASE_STATE.NOTOP, E_RS_BASE_SUBSTATE.NOTOP_NOTREADY);
	RETURN;
END_IF
END_METHOD

END_FUNCTION_BLOCK

// ---- POUs/Pumps/FB_CRYO_PUMP_MVP030.TcPOU
FUNCTION_BLOCK FB_CRYO_PUMP_MVP030 EXTENDS FB_CRYO_PUMP_SERIAL
VAR_INPUT
END_VAR
VAR_OUTPUT
END_VAR
VAR
	
	{attribute 'OPC.UA.DA' := '1'}
	cfg:		T_CRYO_PUMP_MVP030_CFG;	
	{attribute 'OPC.UA.DA' := '1'}
	ctrl:		T_CRYO_PUMP_BASE_CTRL;	
	{attribute 'OPC.UA.DA' := '1'}
	{attribute 'OPC.UA.DA.Access' := '1'}
	stat:		T_CRYO_PUMP_MVP030_STAT;	


	// Input signals
	i_bReady		AT %I*:	BOOL;	// Turbo Pump Ready (signal DO1)
	i_bError		AT %I*:	BOOL;	// If FALSE, Error present - active low (signal DO2)

	// Output signals q_bStart already defined in FB_CRYO_TMP_BASE.
	// q_bStart should activate a relay that 
	// connects Pin 7 with Pin 5 - DI Pumping station

END_VAR


// Execute the base class object FB_CRYO_PUMP_SERIAL
SUPER^();

METHOD M_Configure
VAR_INPUT
END_VAR
VAR
	//
	// List of INIT commands.
	//
	cmdList_Init_MVP030:	ARRAY [1..8] OF T_CRYO_PUMP_CMD := [
		(cmd := cfg.C_CMD_sCtrlViaInt, 		length := 17),	// Reply of 17 chars with the terminator!	
		(cmd := cfg.C_CMD_sFwVersion, 		length := 20),	
		(cmd := cfg.C_CMD_sHwVersion, 		length := 20),
		(cmd := cfg.C_CMD_nNominalSpeed,	length := 20),
		(cmd := '', 						length := 0),
		(cmd := '', 						length := 0),
		(cmd := '', 						length := 0),
		(cmd := '', 						length := 0)];

	//
	//	List of READ (and WRITE) commands.
	// NOTE: Monitoring loop stops on first cmd = ''.
	//
	cmdList_Read_MVP030:	ARRAY [1..16] OF T_CRYO_PUMP_CMD := [
		(cmd := cfg.C_CMD_bON, 				length := 20),	// Reply of 20 chars with the terminator!	
		(cmd := cfg.C_CMD_nCtrlMode, 		length := 17),	
		(cmd := cfg.C_CMD_sErrorCode, 		length := 20),
		(cmd := cfg.C_CMD_nMotorCurr, 		length := 20),
		(cmd := cfg.C_CMD_nPumpHours, 		length := 20),
		(cmd := cfg.C_CMD_nMotorVolt, 		length := 20),
		(cmd := cfg.C_CMD_nElecPower, 		length := 20),
		(cmd := cfg.C_CMD_nPumpTemp, 		length := 20),
		(cmd := cfg.C_CMD_nPumpSpeed, 		length := 20),
		(cmd := '', 						length := 0),
		(cmd := '', 						length := 0),
		(cmd := '', 						length := 0),
		(cmd := '', 						length := 0),
		(cmd := '', 						length := 0),
		(cmd := '', 						length := 0),
		(cmd := '', 						length := 0)];
	
		i:	INT;
END_VAR
IF NOT bStarted	THEN
	//
	// START: Mandatory for ALL pumps !!!
	//
	// Set references from FB_RS_BASE
	cfgRef	REF=cfg;
	ctrlRef	REF=ctrl;
	statRef	REF=stat;

	// Set references from FB_CRYO_TMP_BASE
	cfgBaseRef	REF=cfg;
	ctrlBaseRef	REF=ctrl;
	statBaseRef	REF=stat;
	
	// Copy input parameters to configuration
	cfg.nModel			:= in_nModel;
	cfg.bAutoMonitor	:= in_bAutoMonitor;
	cfg.tDelay_Periodic	:= DINT_TO_TIME(in_nPeriod);
	
	
	// Set pointers to arrays of commands
	ptrInitCmds	:= ADR(cfg.cmdList_Init);(* Pointer to INIT commands *)
	ptrReadCmds	:= ADR(cfg.cmdList_Read);(* Pointer to READ commands *)
	
	// TODO in FB that extends the functionality
	// Set pointers to comm, i.e.
	ptrCommCfg	:= ADR(comm.cfg);	(* Pointer to comm.cfg instance *)
	ptrCommCtrl	:= ADR(comm.ctrl);	(* Pointer to comm.ctrl instance *)
	ptrCommStat	:= ADR(comm.stat);	(* Pointer to comm.stat instance *)
	
	// Set comm suffixes for commands and replies
	ptrCommCfg^.sCmdSuffix		:= in_sCmdSuffix;
	ptrCommCfg^.sReplySuffix	:= in_sReplySuffix;

	statRef.bConfigured	:= TRUE;
	bStarted			:= TRUE;
	//
	// END: Mandatory for ALL pumps !!!
	//


	//
	// ATH specific configuration
	//
	
	// Assign INIT and READ commands.
	cfg.cmdList_Init	:= cmdList_Init_MVP030;
	cfg.cmdList_Read	:= cmdList_Read_MVP030;
	
	// Add checksum to all INIT and READ commands
	FOR i:=1 TO 8 DO
		IF cfg.cmdList_Init[i].cmd <> '' THEN
			cfg.cmdList_Init[i].cmd	:= M_PVP_Checksum(cfg.cmdList_Init[i].cmd);
		ELSE
			EXIT;
		END_IF
	END_FOR
	
	FOR i:=1 TO 16 DO
		IF cfg.cmdList_Read[i].cmd <> '' THEN
			cfg.cmdList_Read[i].cmd	:= M_PVP_Checksum(cfg.cmdList_Read[i].cmd);
		ELSE
			EXIT;
		END_IF
	END_FOR
	
END_IF
END_METHOD

METHOD M_GetSpeed : DINT
VAR_INPUT
END_VAR
M_GetSpeed	:= stat.nPumpSpeed;
END_METHOD

METHOD M_IsReady : BOOL
VAR_INPUT
END_VAR
M_IsReady	:= stat.bReady;
END_METHOD

METHOD M_IsRunning : BOOL
VAR_INPUT
END_VAR
M_IsRunning	:= stat.bMoving;
END_METHOD

METHOD M_ReadFromReply : BOOL
// Method to check correctness of the reply and assign the result to a status variable.
VAR_INPUT
	idx:		INT;		(* arr [idx] will hold the first extracted value, arr [idx+1] the second one, etc. *)
	bInitCmd:	BOOL := FALSE;
END_VAR
VAR
	pos:	INT;
	cmd:	STRING;
	length:	DINT;
	subStr:	STRING;
	valLen:	INT;		// Number of character for the value
END_VAR
// During INIT it might happen that the command index is 0.
// These cases should be discarded.
IF idx <= 0	THEN
	M_ReadFromReply	:= TRUE;
	RETURN;
END_IF

IF bInitCmd	THEN
	cmd		:= cfg.cmdList_Init[idx].cmd;
	length	:= cfg.cmdList_Init[idx].length;
ELSE
	cmd		:= cfg.cmdList_Read[idx].cmd;
	length	:= cfg.cmdList_Read[idx].length;
END_IF

IF length <> 0  AND  LEN(stat.sReply) <> length THEN
	stat.sErrorText	:= 'Wrong reply length';
	M_ReadFromReply	:= FALSE;
	RETURN;
END_IF

// Check if sent command was correct.
IF	FIND(stat.sReply,'NO_DEF') > 0	OR 
	FIND(stat.sReply,'_RANGE') > 0	OR 
	FIND(stat.sReply,'_LOGIC') > 0		THEN
	// Wrong command sent. This is an error.
	stat.sErrorText	:= 'Incorrect command';
	M_ReadFromReply	:= FALSE;
	RETURN;
END_IF

// Check the structure of the reply.
// Example 1 - Data query with 6 characters for the value:
//    CMD:   1 2 3 0 0 3 0 9 0 2 = ? 1 1 2 cR
//    Reply: 1 2 3 1 0 3 0 9 0 6 0 0 0 6 3 3 0 3 7 cR
//    valLen = 6 (from '06' in reply)
//    value = 633
// Example 2 - Data query with 3 characters for the value:
//    CMD:   1 2 3 0 0 0 6 0 0 2 = ? x x x cR
//    Reply: 1 2 3 1 0 0 6 0 0 3 0 0 2 y y y cR
//    valLen = 3 (from '03' in reply)
//    value = 002 = 2
// Example 3 - Command (reply is identical to command):
//    CMD:   0 4 2 1 0 0 1 0 0 6 1 1 1 1 1 1 0 2 0 cR
//    Reply: 0 4 2 1 0 0 1 0 0 6 1 1 1 1 1 1 0 2 0 cR
//    valLen = 6 (from '06' in reply)
//
// Compared to the first 10 chars of the command, 
// the reply should modify characters 3 and 9 (index starts from 0)
// reply[3] = 1
// reply[9] = length - 14
//
// So, we want to convert: 1 2 3 0 0 3 0 9 0 2
//                     to: 1 2 3 1 0 3 0 9 0 6
// Extract first 10 characters from the command
subStr	:= MID(cmd,10,1);
// Replace character [3] with '1', i.e. with ASCII 49.
subStr[3]	:= 49;
// Replace character [9] with expected number of characters in the value.
valLen	:= DINT_TO_INT(length - 14);
// Convert integer to character.
subStr[9]	:= INT_TO_BYTE(valLen + 48);
IF	FIND(stat.sReply,subStr) <> 1	THEN
	// Wrong reply received. This is an error.
	stat.sErrorText	:= 'Wrong reply received';
	M_ReadFromReply	:= FALSE;
	RETURN;
END_IF


//
// All fine so far. Let's extract the reading.
//
// The actual reply is contained in the 'valLen' (3 or 6) characters starting 
// from char [10] (11-the character for MID() function).
subStr	:= MID(stat.sReply, valLen, 11);

// Remove the 3-character checksum from the command.
cmd	:= MID(cmd, LEN(cmd)-3,1);

IF cmd = cfg.C_CMD_sFwVersion	THEN
	stat.sFwVersion		:= MID(subStr, 6, 1);
ELSIF cmd = cfg.C_CMD_sHwVersion	THEN
	stat.sHwVersion		:= MID(subStr, 6, 1);
ELSIF cmd = cfg.C_CMD_nNominalSpeed	THEN
	stat.nNominalSpeed	:= LREAL_TO_DINT(STRING_TO_LREAL(subStr));		// [rpm]
ELSIF cmd = cfg.C_CMD_bON	THEN
	stat.bON	:= STRING_TO_BOOL(subStr) <> FALSE;
ELSIF cmd = cfg.C_CMD_nCtrlMode	THEN
	stat.nCtrlMode	:= STRING_TO_DINT(subStr);
ELSIF cmd = cfg.C_CMD_sErrorCode	THEN
	IF	FIND(subStr,'Err') > 0	OR 
		FIND(subStr,'Wrn') > 0		THEN
		// There is an Error or Warning.
		stat.sFailureCode	:= MID(subStr, 6, 1);
		stat.bFailure		:= TRUE;
	ELSE
		stat.sFailureCode	:= 'OK';
		stat.bFailure		:= FALSE;
	END_IF
ELSIF cmd = cfg.C_CMD_nMotorCurr	THEN
	stat.nMotorCurr	:= STRING_TO_DINT(subStr) * 10;		// [mA]
ELSIF cmd = cfg.C_CMD_nPumpHours	THEN
	stat.nPumpHours	:= STRING_TO_DINT(subStr);
ELSIF cmd = cfg.C_CMD_nMotorVolt	THEN
	stat.nMotorVolt	:= STRING_TO_DINT(subStr) / 100;	// [V]
	stat.lrMotorVolt:= STRING_TO_LREAL(subStr) / 100.0;	// [V]
ELSIF cmd = cfg.C_CMD_nElecPower	THEN
	stat.nElecPower	:= STRING_TO_DINT(subStr);			// [W]
ELSIF cmd = cfg.C_CMD_nPumpTemp	THEN
	stat.nPumpTemp	:= STRING_TO_DINT(subStr);			// [°C]
ELSIF cmd = cfg.C_CMD_nPumpSpeed	THEN
	stat.nPumpSpeed	:= LREAL_TO_DINT(STRING_TO_LREAL(subStr));			// [rpm]
END_IF


M_ReadFromReply	:= TRUE;	// OK
END_METHOD

METHOD M_UpdateStatus
VAR_INPUT
END_VAR
// Update Status from digital inputs readings
stat.bReady		:= i_bReady;
stat.bFailure	:= NOT i_bError;	// Active low

stat.bMoving	:= stat.bReady OR stat.nPumpSpeed > 0;

// Set Control Mode Label
(*
	1 = remote
	2 = RS-485
	4 = PV.can
	32 = Keys on the front panel
*)
CASE stat.nCtrlMode	OF
	1:		stat.sCtrlMode	:= 'REMOTE';
	2:		stat.sCtrlMode	:= 'RS-485';
	4:		stat.sCtrlMode	:= 'PV.can';
	32:		stat.sCtrlMode	:= 'Keys on Front Panel';
ELSE
	stat.sCtrlMode	:= 'UNKNOWN';
END_CASE
END_METHOD

END_FUNCTION_BLOCK

// ---- POUs/Pumps/FB_CRYO_PUMP_SERIAL.TcPOU
// Cryo Turbo Molecular Pump Control
FUNCTION_BLOCK FB_CRYO_PUMP_SERIAL EXTENDS FB_CRYO_PUMP_BASE
VAR_INPUT
	{attribute 'OPC.UA.DA' := '0'}
	in_sCmdSuffix:		STRING(16) := '$0D';
	{attribute 'OPC.UA.DA' := '0'}
	in_sReplySuffix:	STRING(16) := '$0D';
END_VAR
VAR_OUTPUT
END_VAR
VAR

	{attribute 'OPC.UA.DA' := '0'}
	comm:		FB_RS_COMM_NO_SIM;			// No simulation yet
	
	// Pointers to structures inside FB_RS_COMM, e.g. ptrCommCfg.
	{attribute 'OPC.UA.DA' := '0'}
	ptrCommCfg:		POINTER TO T_RS_COMM_CFG;	(* Pointer to comm.cfg instance *)
	{attribute 'OPC.UA.DA' := '0'}
	ptrCommCtrl:	POINTER TO T_RS_COMM_CTRL;	(* Pointer to comm.ctrl instance *)
	{attribute 'OPC.UA.DA' := '0'}
	ptrCommStat:	POINTER TO T_RS_COMM_STAT;	(* Pointer to comm.stat instance *)

END_VAR

// Execute the base class object FB_RS_BASE
SUPER^();

METHOD ActivityInitializing
VAR_INPUT
	bExecute:	BOOL;
END_VAR
VAR_INST
	{attribute 'OPC.UA.DA' := '0'}
    nMethodState:	INT := 0;	// State Machine current state
END_VAR
SetAction('ActivityInitializing');


IF NOT bExecute THEN
	nMethodState	:= 0;	// Reset the state machine
	cmdCounter		:= 0;	// Init will start from the first init command after increment
	RETURN;
END_IF

// Handle State Machine
CASE nMethodState OF
	0:	// Set initial state and status
		statRef.bInitialised	:= FALSE;
		statBaseRef.sReply			:= '';
		SetStatus(E_SM_ERROR.OK, 'BUSY');

		nMethodState := 10;				// Go to next state, i.e. INIT_COMM

	10:	// Initialize COMM port
		(* Reset the serial port *)
		ptrCommCtrl^.nCommand	:= E_RS_COMM_CMD.INIT;
		ptrCommCtrl^.bExecute	:= TRUE;

		(* Start the timer by going false/true *)
		fbTimer (IN := FALSE); (* Reset timer *)
		fbTimer (IN := TRUE, PT := T#5S); (* 5 sec timeout for reply *)

		nMethodState 	:= 15;	// On next cycle wait until the comm port is reset, i.e. idle
		
	15:	// Wait IDLE
		fbTimer (IN := TRUE);
		IF comm.stat.nStatus = E_RS_COMM_STATUS.IDLE THEN
			// Communication is IDLE 
			fbTimer (IN := FALSE);	// disable timer 
			statBaseRef.sReply		:= ptrCommStat^.sReply;	// Save the reply

			// TODO Assign the value to a status variable.
			IF NOT M_ReadFromReply(cmdCounter, TRUE)	THEN
				cmdCounter		:= 0;	// Reset command counter
				nMethodState 	:= 10;	// Wait for INIT
			ELSE
				cmdCounter		:= cmdCounter + 1;	// Increment init command index
				fbTimer (IN := FALSE);	// disable timer 
				fbTimer (IN := TRUE, PT := cfgRef.tDelay_Init); // Wait INIT delay
				bCommProblem	:= FALSE;
				nMethodState 	:= 18;	// Execute next device INIT command
			END_IF
		ELSIF comm.stat.nStatus = E_RS_COMM_STATUS.ERROR THEN
			fbTimer (IN := FALSE);
			SetStatus(E_LAKESHORE_ERROR.COMM, 'ERROR: Communication error');	
			bCommProblem	:= TRUE;
			nEvent := E_SM_EVENT.ERRINIT;
			RETURN;
		ELSIF fbTimer.Q THEN
			// Timer expired after 5 sec. This is an error.
			fbTimer (IN := FALSE);
			SetStatus(E_LAKESHORE_ERROR.TIMEOUT, 'ERROR: Communication timeout');	
			bCommProblem	:= TRUE;
			nEvent := E_SM_EVENT.ERRINIT;
			RETURN;
		END_IF

	
	
	18:	// Wait INIT Delay
		fbTimer (IN := TRUE);
		IF fbTimer.Q THEN
			// Timer expired after 5 sec. This is an error.
			fbTimer (IN := FALSE);
			nMethodState 	:= 20;	// Execute next device INIT command
			RETURN;
		END_IF

	
	
	20:	// INIT DEV
		IF ptrInitCmds^ [cmdCounter].cmd = '' THEN
			// Device INIT is done. Go to IDLE 
			statRef.bInitialised 	:= TRUE;
			cmdCounter			:= 1;
			SetStatus(E_SM_ERROR.OK, 'IDLE');
			nEvent 		:= E_SM_EVENT.INITDONE;
			RETURN;
		END_IF
		
		(* Send INIT command with index cmdCounter *)
		ptrCommCtrl^.nCommand		:= E_RS_COMM_CMD.SEND;
		ptrCommCtrl^.sCmd			:= ptrInitCmds^ [cmdCounter].cmd;
		ptrCommCtrl^.nNumReplies	:= 1;
		ptrCommCtrl^.bHasReply		:= TRUE;
		ptrCommCtrl^.bExecute		:= TRUE;
	
		(* Start the timer by going false/true *)
		fbTimer (IN := FALSE); (* Reset timer *)
		fbTimer (IN := TRUE, PT := T#5S); (* 5 sec timeout for reply *)

		// On next cycle wait until the comm port is idle
		nMethodState 	:= 15;	// On next cycle wait until the comm port is idle
	
END_CASE
END_METHOD

METHOD ActivityMonitoring
VAR_INPUT
	bExecute:	BOOL;
END_VAR
VAR_INST
	{attribute 'OPC.UA.DA' := '0'}
    nMethodState:	INT := 0;	// State Machine current state
	{attribute 'OPC.UA.DA' := '0'}
	nRetries:		INT := 0;	// Number of retries in case of communication problems
END_VAR

VAR
	offset: INT;
END_VAR
IF NOT cfgRef.bAutoMonitor AND statRef.nSubstate = E_RS_BASE_SUBSTATE.NOTOP_READY THEN
	SetAction('No Monitoring'); 
	SetStatus(E_SM_ERROR.OK, 'IDLE');
	nMethodState	:= 0;	// Reset the state machine
	cmdCounter		:= 1;	// Reading will start from the first command in the array
	RETURN;
END_IF

IF NOT bExecute THEN
	SetAction('ActivityMonitoring'); 
	SetStatus(E_SM_ERROR.OK, 'BUSY');
	nMethodState	:= 0;	// Reset the state machine
	cmdCounter		:= 1;	// Reading will start from the first command in the array
	RETURN;
END_IF

// Handle State Machine
CASE nMethodState OF
	0:	// Execute a command from the command array
		IF ptrReadCmds^ [cmdCounter].cmd = '' OR cmdCounter > 16 THEN

			// All commands have been executed. 
			// Wait tDelay_Periodic before re-starting the READ.
			cmdCounter	:= 1;
			SetStatus(E_SM_ERROR.OK, 'IDLE');
			
			(* Start the timer by going false/true *)
			fbTimer (IN := FALSE); (* Reset timer *)
			fbTimer (IN := TRUE, PT := cfgRef.tDelay_Periodic);
			nMethodState := 10;				// Goto Wait for tDelay_Periodic
			RETURN;
			
		END_IF
		
		(* Send command with index cmdCounter *)
		ptrCommCtrl^.nCommand		:= E_RS_COMM_CMD.SEND;
		ptrCommCtrl^.sCmd			:= ptrReadCmds^ [cmdCounter].cmd;
		ptrCommCtrl^.nNumReplies	:= 1;
		ptrCommCtrl^.bHasReply		:= TRUE;
		ptrCommCtrl^.bExecute		:= TRUE;
		
		// In case we are executing 'SET' commands, there are no replies.
		// However, we need a delay of at least 50ms between commands.
		// We will apply 150ms.
		IF NOT ptrCommCtrl^.bHasReply THEN
			// There is no reply, i.e. this is a 'SET' command.
			// Start the timer by going false/true.
			// Apply 200ms delay between SET commands.
			fbTimer (IN := FALSE); // Reset timer
			fbTimer (IN := TRUE, PT := T#200MS); 
			cmdCounter		:= cmdCounter + 1;	// Go to next command.
			nMethodState	:= 10;				// Goto WAIT for Reading to complete,
			RETURN;
		ELSE			
			// There is a reply, i.e. this is a 'READ' command.
			// Apply short delay of 10ms before checking the status. 
			// Start the timer by going false/true
			fbTimer (IN := FALSE); // Reset timer
			fbTimer (IN := TRUE, PT := T#10MS);	
			statRef.sErrorText	:= 'BUSY';
			nMethodState := 15;	// Goto WAIT for Reading to complete,
		END_IF
		

	10:	// Wait until the delay timeout expires
		fbTimer (IN := TRUE);

		(* If Timer has expired, go to the next state. *)
		IF fbTimer.Q THEN
			fbTimer (IN := FALSE);
			nMethodState 	:= 0;	// Goto Wait for tDelay_Periodic
			RETURN;
		END_IF
	
	15:	// Wait until the delay timeout expires
		fbTimer (IN := TRUE);

		(* If Timer has expired, go to the next state. *)
		IF fbTimer.Q THEN
			fbTimer (IN := FALSE);
			fbTimer (IN := TRUE, PT := T#5S);	// 5 sec timeout for reply
			statRef.sErrorText	:= 'BUSY';
			nMethodState 	:= 20;	// Goto Wait for IDLE/Reply
			RETURN;
		END_IF
	



	20:	// Wait for the reading to complete, i.e. IDLE
		fbTimer (IN := TRUE);
		IF comm.stat.nStatus = E_RS_COMM_STATUS.IDLE THEN
			// Communication is IDLE 
			fbTimer (IN := FALSE);	// disable timer 
			statBaseRef.sReply		:= ptrCommStat^.sReply;	// Save the reply
			
			// Copy readings to status variable(s)
			
			// TODO Assign the value to a status variable.
			IF NOT M_ReadFromReply(cmdCounter, FALSE)	THEN
				// Reply was not OK. Maybe out of sync.
				// Re-INIT the communication, i.e. clear the buffer.
				ptrCommCtrl^.nCommand	:= E_RS_COMM_CMD.INIT;
				ptrCommCtrl^.bExecute	:= TRUE;
		
				(* Start the timer by going false/true *)
				fbTimer (IN := FALSE); (* Reset timer *)
				fbTimer (IN := TRUE, PT := T#5S); (* 5 sec timeout for reply *)
		
				SetStatus(E_LAKESHORE_ERROR.COMM, 'ERROR: Communication error');	
				bCommProblem	:= TRUE;

				nMethodState 	:= 10;	// On next cycle wait until the comm port is reset, i.e. idle
				RETURN;
			ELSE
				// All OK. Go to next command.
				bCommProblem	:= FALSE;
				nRetries		:= 0;	// Reset number of retries
		
				cmdCounter		:= cmdCounter + 1;	// Go to next command.
				
				// Apply a 50 ms delay between commands
				fbTimer (IN := FALSE);	// Reset timer
				fbTimer (IN := TRUE, PT := T#50MS); 
				nMethodState := 10;		// Apply delay
				nEvent := E_SM_EVENT.COMMOK;
				RETURN;
			END_IF
		ELSIF comm.stat.nStatus = E_RS_COMM_STATUS.ERROR OR fbTimer.Q THEN
			// No Reply.
			// Re-INIT the communication, i.e. clear the buffer.
			ptrCommCtrl^.nCommand	:= E_RS_COMM_CMD.INIT;
			ptrCommCtrl^.bExecute	:= TRUE;
	
			(* Start the timer by going false/true *)
			fbTimer (IN := FALSE); (* Reset timer *)
			fbTimer (IN := TRUE, PT := T#5S); (* 5 sec timeout for reply *)
	
			SetStatus(E_LAKESHORE_ERROR.COMM, 'ERROR: Communication error');	
			bCommProblem	:= TRUE;

			nRetries		:= nRetries + 1;		// Increment number of retries
			statBaseRef.nRetries	:= statBaseRef.nRetries + 1;	// Increment total number of retries

			nMethodState 	:= 10;	// On next cycle wait until the comm port is reset, i.e. idle
			RETURN;
		END_IF

	
END_CASE
END_METHOD

METHOD M_ExecuteComm
VAR_INPUT
END_VAR
comm(in_sCmdSuffix:=in_sCmdSuffix, in_sReplySuffix:=in_sReplySuffix, in_nTimeout:=3000);
END_METHOD

METHOD M_GetCouplerState : BOOL
VAR_INPUT
END_VAR
IF comm.i_nCouplerState = 8 THEN
	M_GetCouplerState	:= TRUE;	
ELSE
	M_GetCouplerState	:= FALSE;	
END_IF
END_METHOD

// Add checksum at the end of Pfeiffer Vacuum Protocol (PVP) command
METHOD M_PVP_Checksum : STRING(24)
VAR_INPUT
	sCmd:	STRING;	// Command without the checksum
END_VAR
VAR
	i:			INT;
	nVar:		SINT;
	nSum:		INT;
	nRes:		INT;	// Resulting check sum
	sCmdFull:	STRING(24);	// Command with the checksum
    fbFormat:	FB_FormatString;
	sTmp:		T_MaxString;
	length:		INT;
END_VAR
// Get the command length
length	:= LEN(sCmd);

nSum	:= 0;
FOR i:=0 TO (length-1) DO
	nSum	:= nSum + BYTE_TO_SINT(sCmd[i]);
END_FOR
nRes	:= nSum MOD 256;

sTmp	:= sCmd;
fbFormat(	sFormat := '%s%.3d', 
			arg1 := F_STRING(sTmp), 
			arg2 := F_INT(nRes), 
			sOut => sCmdFull);
			
M_PVP_Checksum	:= sCmdFull;
END_METHOD

METHOD M_ReadFromReply : BOOL
// Method to check correctness of the reply and assign the result to a status variable.
VAR_INPUT
	idx:		INT;		(* arr [idx] will hold the first extracted value, arr [idx+1] the second one, etc. *)
	bInitCmd:	BOOL := FALSE;
END_VAR
VAR
	pos:	INT;
	cmd:	STRING;
	length:	DINT;
	subStr:	STRING(255);
END_VAR
// TODO: Implement specific parsing of replies
END_METHOD

END_FUNCTION_BLOCK

// ---- POUs/Pumps/FB_CRYO_PUMP_HIPACE30.TcPOU
FUNCTION_BLOCK FB_CRYO_PUMP_HIPACE30 EXTENDS FB_CRYO_PUMP_SERIAL
VAR_INPUT
END_VAR
VAR_OUTPUT
END_VAR
VAR
	
	{attribute 'OPC.UA.DA' := '1'}
	cfg:		T_CRYO_PUMP_HIPACE30_CFG;	
	{attribute 'OPC.UA.DA' := '1'}
	ctrl:		T_CRYO_PUMP_BASE_CTRL;	
	{attribute 'OPC.UA.DA' := '1'}
	{attribute 'OPC.UA.DA.Access' := '1'}
	stat:		T_CRYO_PUMP_HIPACE30_STAT;	


	// Input signals
	i_bReady		AT %I*:	BOOL;	// Turbo Pump Ready (signal DO1)
	i_bError		AT %I*:	BOOL;	// If FALSE, Error present - active low (signal DO2)

	// Output signals q_bStart already defined in FB_CRYO_TMP_BASE.
	// q_bStart should activate a relay that 
	// connects Pin 7 with Pin 5 - DI Pumping station

END_VAR


// Execute the base class object FB_CRYO_PUMP_SERIAL
SUPER^();

METHOD M_Configure
VAR_INPUT
END_VAR
VAR
	//
	// List of INIT commands.
	//
	cmdList_Init_HIPACE30:	ARRAY [1..8] OF T_CRYO_PUMP_CMD := [
		(cmd := cfg.C_CMD_sCtrlViaInt, 		length := 17),	// Reply of 17 chars with the terminator!	
		(cmd := cfg.C_CMD_sFwVersion, 		length := 20),	
		(cmd := cfg.C_CMD_sHwVersion, 		length := 20),
		(cmd := cfg.C_CMD_nNominalSpeed,	length := 20),
		(cmd := '', 						length := 0),
		(cmd := '', 						length := 0),
		(cmd := '', 						length := 0),
		(cmd := '', 						length := 0)];

